	            // Check gaps is a routine that checks all the time if the gap and head to head distance is acording to the configuration.
	            // If not, the bit "sx_Gapping" is set true and the conveyor stops to gap.
	            // Compare gaps calculated with the configured gaps
	            IF NOT #sx_ReverseDirection
	            THEN
	                REGION 7.5.1 - Forward

	                    IF ((#sdi_GapHeadToHeadConfigurationFwd > #sdi_GapHeadToHeadFwd               // Compare head to head configured with real distance
	                        OR #sdi_GapTailToHeadConfigurationFwd > #sdi_GapFwd
	                        OR #sdi_GapTailToHeadConfigurationFwd > #sdi_DownstreamGapTailtoHeadFwd           // Compare gap configured with real gap
	                        OR #sdi_GapHeadToHeadConfigurationFwd > #sdi_DownstreamGapHeadToHeadFwd)
	                        AND #sF_TRIG_AuxHeadToEnd_Fwd.Q)                                                         // Trigger when parcel arrive in the end of the conveyor
	                    THEN

	                        #sx_GappingFwd := TRUE;        // Bit to inform the system that conveyor needs to stop to apply gap

	                    END_IF;

	                END_REGION
	            ELSE
	                REGION 7.5.1 - Reverse

	                    IF ((#sdi_GapHeadToHeadConfigurationRvs > #sdi_GapHeadToHeadRvs               // Compare head to head configured with real distance
	                        OR #sdi_GapTailToHeadConfigurationRvs > #sdi_Gap_Rvs
	                        OR #sdi_GapTailToHeadConfigurationRvs > #sdi_DownstreamGapTailtoHeadRvs           // Compare gap configured with real gap
	                        OR #sdi_GapHeadToHeadConfigurationRvs > #sdi_DownstreamGapHeadToHeadRvs)
	                        AND #sF_TRIG_AuxHeadToEnd_Rvs.Q)                                                         // Trigger when parcel arrive in the end of the conveyor
	                    THEN

	                        #sx_GappingRvs := TRUE;        // Bit to inform the system that conveyor needs to stop to apply gap

	                    END_IF;

	                END_REGION
	            END_IF;
	            //    When conveyor stops to gapping, displacement values from downstream are used to
	            //    apply new gap.
	            //    When the new gap applied fits with the configured one, the conveyor starts running again.
	            //    If the conveyor stops for die back reason and the gap its been applied, and extra gap value it will be applied.
	            //    This recovery gap it helps to recovery the system after die back.
	            IF NOT #sx_ReverseDirection
	            THEN
	                REGION 7.5.3 - Forward

	                    IF (#sx_GappingFwd          // Gapping needs to be applied bit
	                        AND ((#sdi_GapHeadToHeadConfigurationFwd > #sdi_GapHeadToHeadFwd    // Configured head to head bigger than the actual one
	                        OR #sdi_GapHeadToHeadConfigurationFwd - #idi_PECEoSDistance / 10 + #sdi_PECtoEndDistanceFwd > #sdi_DownstreamGapHeadToHeadFwd
	                        OR #sdi_GapTailToHeadConfigurationFwd > #sdi_GapFwd     // Configured gap bigger than the actual one
	                        OR #sdi_GapTailToHeadConfigurationFwd - #idi_PECEoSDistance / 10 + #sdi_PECtoEndDistanceFwd > #sdi_DownstreamGapTailtoHeadFwd)
	                        AND NOT #sx_RecoveryGapFwd)                                                // Die back recovery gap bit not active
	                        OR (((#sdi_GapHeadToHeadConfigurationFwd + #iUDT_ConveyorConfiguration.ExtraGapRecovery)   // Add recovery gap to the configured
	                        > #sdi_GapHeadToHeadFwd                                                                                 // Actual head to head distance
	                        OR (#sdi_GapHeadToHeadConfigurationFwd - #idi_PECEoSDistance / 10 + #sdi_PECtoEndDistanceFwd + #iUDT_ConveyorConfiguration.ExtraGapRecovery)
	                        > #sdi_DownstreamGapHeadToHeadFwd
	                        OR (#sdi_GapTailToHeadConfigurationFwd + #iUDT_ConveyorConfiguration.ExtraGapRecovery)    // Add recovery gap to the configured
	                        > #sdi_GapFwd                                                                               // Actual gap between parcels
	                        OR (#sdi_GapTailToHeadConfigurationFwd - #idi_PECEoSDistance / 10 + #sdi_PECtoEndDistanceFwd + #iUDT_ConveyorConfiguration.ExtraGapRecovery)
	                        > #sdi_DownstreamGapTailtoHeadFwd)
	                        AND #sx_RecoveryGapFwd))                                                                       // Recovery gap bit activate
	                    THEN

	                        #sdi_GapHeadToHeadFwd += #iqUDT_HandShake.DownstreamDisplacement;      // Increase head to head counter with conveyor downstream displacement
	                        #sdi_GapFwd += #iqUDT_HandShake.DownstreamDisplacement;     // Increase gap counter with conveyor downstream displacement

	                    ELSE

	                        #sx_GappingFwd := FALSE;                   // Set gapping bit to false

	                    END_IF;

	                    IF #sx_GappingFwd                              // Gapping bit active
	                        AND NOT #iqUDT_HandShake.RTR           // Ready to receive not active
	                    THEN

	                        #sx_RecoveryGapFwd := TRUE;                // Recovery gap activation after die back

	                    END_IF;

	                    IF #sx_RecoveryGapFwd                          // Recovery gap active
	                        AND NOT #sx_GappingFwd                     // Gapping bit not active
	                    THEN

	                        #sx_RecoveryGapFwd := FALSE;               // Recovery gap disable

	                    END_IF;

	                END_REGION
	            ELSE
	                REGION 7.5.4 - Reverse

	                    IF (#sx_GappingRvs          // Gapping needs to be applied bit
	                        AND ((#sdi_GapHeadToHeadConfigurationRvs > #sdi_GapHeadToHeadRvs    // Configured head to head bigger than the actual one
	                        OR #sdi_GapHeadToHeadConfigurationRvs - #idi_PECBoSDistance / 10 + #sdi_PECtoEndDistanceRvs > #sdi_DownstreamGapHeadToHeadRvs
	                        OR #sdi_GapTailToHeadConfigurationRvs > #sdi_Gap_Rvs     // Configured gap bigger than the actual one
	                        OR #sdi_GapTailToHeadConfigurationRvs - #idi_PECBoSDistance / 10 + #sdi_PECtoEndDistanceRvs > #sdi_DownstreamGapTailtoHeadRvs)
	                        AND NOT #sx_RecoveryGapRvs)                                                // Die back recovery gap bit not active
	                        OR (((#sdi_GapHeadToHeadConfigurationRvs + #iUDT_ConveyorConfiguration.ExtraGapRecovery)   // Add recovery gap to the configured
	                        > #sdi_GapHeadToHeadRvs                                                                                 // Actual head to head distance
	                        OR (#sdi_GapHeadToHeadConfigurationRvs - #idi_PECBoSDistance / 10 + #sdi_PECtoEndDistanceRvs + #iUDT_ConveyorConfiguration.ExtraGapRecovery)
	                        > #sdi_DownstreamGapHeadToHeadRvs
	                        OR (#sdi_GapTailToHeadConfigurationRvs + #iUDT_ConveyorConfiguration.ExtraGapRecovery)    // Add recovery gap to the configured
	                        > #sdi_Gap_Rvs                                                                               // Actual gap between parcels
	                        OR (#sdi_GapTailToHeadConfigurationRvs - #idi_PECBoSDistance / 10 + #sdi_PECtoEndDistanceRvs + #iUDT_ConveyorConfiguration.ExtraGapRecovery)
	                        > #sdi_DownstreamGapTailtoHeadRvs)
	                        AND #sx_RecoveryGapRvs))                                                                                // Recovery gap bit activate
	                    THEN

	                        #sdi_GapHeadToHeadRvs -= #iqUDT_HandShakeUp.DownstreamDisplacement;      // Increase head to head counter with conveyor downstream displacement
	                        #sdi_Gap_Rvs -= #iqUDT_HandShakeUp.DownstreamDisplacement;     // Increase gap counter with conveyor downstream displacement

	                    ELSE

	                        #sx_GappingRvs := FALSE;                   // Set gapping bit to false

	                    END_IF;

	                    IF #sx_GappingRvs                              // Gapping bit active
	                        AND NOT #iqUDT_HandShakeUp.RTR           // Ready to receive not active
	                    THEN

	                        #sx_RecoveryGapRvs := TRUE;                // Recovery gap activation after die back

	                    END_IF;

	                    IF #sx_RecoveryGapRvs                          // Recovery gap active
	                        AND NOT #sx_GappingRvs                     // Gapping bit not active
	                    THEN

	                        #sx_RecoveryGapRvs := FALSE;               // Recovery gap disable

	                    END_IF;

	                END_REGION
	            END_IF;
	        END_REGION

	        REGION 7.6 - Ready to send and Transfer in progress
	            IF NOT #sx_ReverseDirection
	            THEN
	                REGION 7.6.1 - Forward

	                    IF #iqUDT_HandShake.RTR                                            // Ready to receive bit
	                        AND NOT #sx_GappingFwd
	                        AND #sx_AuxHeadAtEndFwd                                            // Parcel is at end of conveyor
	                        AND NOT #ix_ExternalRequestDieBack
	                    THEN

	                        #iqUDT_HandShake.TIP := TRUE;      // Transfer in progress bit
	                        #iqUDT_HandShake.RTS := FALSE;     // Ready to send bit
	                        #sx_AuxHeadAtEndFwd := FALSE;

	                    END_IF;

	                    IF #sR_TRIG_TailToBegin_Fwd.Q               // Reset TIP when the parcel leaves interlock
	                    THEN

	                        #iqUDT_HandShake.TIP := FALSE;     // Transfer in progress bit

	                    END_IF;

	                END_REGION
	            ELSE
	                REGION 7.6.2 - Reverse

	                    IF #iqUDT_HandShakeUp.RTR                                            // Ready to receive bit
	                        AND #iqUDT_HandShake.RTR
	                        AND NOT #sx_GappingRvs
	                        AND #sx_AuxHeadAtEndRvs                                            // Parcel is at end of conveyor
	                        AND NOT #ix_ExternalRequestDieBack
	                    THEN

	                        #iqUDT_HandShakeUp.TIP := TRUE;      // Transfer in progress bit
	                        #iqUDT_HandShakeUp.RTS := FALSE;     // Ready to send bit
	                        #sx_AuxHeadAtEndRvs := FALSE;

	                    END_IF;

	                    IF #sR_TRIG_TailToBegin_Rvs.Q               // Reset TIP when the parcel leaves interlock
	                    THEN

	                        #iqUDT_HandShakeUp.TIP := FALSE;     // Transfer in progress bit

	                    END_IF;

	                END_REGION
	            END_IF;
	        END_REGION

	        REGION 7.7 - Downstream gap

	            (* This functionality is used to maintain the gap between parcel conveyor's downstream.
	               To do this, is used the downstream displacement.  *)
	            IF NOT #sx_ReverseDirection
	            THEN
	                REGION 7.7.1 - Forward

	                    IF #sR_TRIG_TailToBegin_Fwd.Q                       // When the parcel's tail reach the beginning of downstream conveyor
	                    THEN

	                        #sdi_DownstreamGapTailtoHeadFwd := 0;                     // Reset downstream gap counter

	                    END_IF;

	                    IF #sdi_DownstreamGapTailtoHeadFwd < #ci_OverflowLimit        // Prevent integer variable overflow
	                    THEN

	                        #sdi_DownstreamGapTailtoHeadFwd += #iqUDT_HandShake.DownstreamDisplacement;          // Downstream displacement gap counter

	                    END_IF;

	                END_REGION
	            ELSE
	                REGION 7.7.2 - Reverse

	                    IF #sR_TRIG_TailToBegin_Rvs.Q                       // When the parcel's tail reach the beginning of downstream conveyor
	                    THEN

	                        #sdi_DownstreamGapTailtoHeadRvs := 0;                     // Reset downstream gap counter

	                    END_IF;

	                    IF #sdi_DownstreamGapTailtoHeadRvs < #ci_OverflowLimit        // Prevent integer variable overflow
	                    THEN

	                        #sdi_DownstreamGapTailtoHeadRvs -= #iqUDT_HandShakeUp.DownstreamDisplacement;          // Downstream displacement gap counter

	                    END_IF;

	                END_REGION
	            END_IF;
	        END_REGION

	        REGION 7.8 - Downstream Head to Head
	            IF NOT #sx_ReverseDirection
	            THEN
	                REGION 7.8.1 - Forward

	                    #sR_TRIG_Transfering_Fwd(CLK := #iqUDT_HandShake.TIP);

	                    IF #sR_TRIG_Transfering_Fwd.Q                                                           // Transfering aux bit rising trigger
	                    THEN

	                        #sdi_DownstreamGapHeadToHeadFwd := 0;                                              // Downstream head to head reset counter

	                    END_IF;

	                    IF #sdi_DownstreamGapHeadToHeadFwd < #ci_OverflowLimit                                 // Prevent integer variable overflow
	                    THEN

	                        #sdi_DownstreamGapHeadToHeadFwd += #iqUDT_HandShake.DownstreamDisplacement;       // Downstream displacement head to head counter

	                    END_IF;

	                END_REGION
	            ELSE
	                REGION 7.8.2 - Reverse

	                    #sR_TRIG_Transfering_Rvs(CLK := #iqUDT_HandShake.TIP);

	                    IF #sR_TRIG_Transfering_Rvs.Q                                                           // Transfering aux bit rising trigger
	                    THEN

	                        #sdi_DownstreamGapHeadToHeadRvs := 0;                                              // Downstream head to head reset counter

	                    END_IF;

	                    IF #sdi_DownstreamGapHeadToHeadRvs < #ci_OverflowLimit                                 // Prevent integer variable overflow
	                    THEN

	                        #sdi_DownstreamGapHeadToHeadRvs -= #iqUDT_HandShakeUp.DownstreamDisplacement;       // Downstream displacement head to head counter

	                    END_IF;

	                END_REGION
	            END_IF;
	        END_REGION

	        REGION 7.9 - Energy save

	            (* Save energy functionality is used to stop conveyor if no parcels are in the system to save energy
	               Save energy function counts displacement if the photo eye do not detects parcels. The counter is reset if:
	               - Photo eye is triggered.
	               - Reset is required from external.
	               - Ready to send is active from upstream. *)

	            IF #iUDT_ConveyorConfiguration.Energy                                       // Energy save functionality enable from configuration
	            THEN

	                IF #sdi_AuxEnergySaveFwd >= #iUDT_ConveyorConfiguration.Forward_Direction.EnergySaveLenght        // Compare energy save counter with configured lenght
	                    OR #sdi_AuxEnergySaveRvs >= #iUDT_ConveyorConfiguration.Reverse_Direction.EnergySaveLenght
	                THEN
	                    #sx_EnergySaveActive := TRUE;                                           // Set energy save active true
	                END_IF;

	                IF ((NOT #ix_PECEoS OR NOT #ix_PECBoS)                                  // Photo eye detects a parcel
	                    AND NOT #sx_EnergySaveActive)                                         // Energy save active bit
	                    OR #ix_ResetEnergySave                                               // Reset energy save
	                    OR (#iqUDT_HandShakeUp.ResetEnergySave AND NOT #sx_ReverseDirection)                               // Reset energy save externaly
	                    OR (#iqUDT_HandShake.ResetEnergySave AND #sx_ReverseDirection)
	                    OR NOT #iqUDT_EquipmentControl.Command.AutomaticOn                  // Automatic ON from control block
	                    OR #iqUDT_EquipmentControl.Command.Stop                             // Stop command from control block
	                THEN
	                    #sdi_AuxEnergySaveFwd := 0;                                        // Reset energy save counter
	                    #sdi_AuxEnergySaveRvs := 0;                                        // Reset energy save counter
	                    #sx_EnergySaveActive := FALSE;                                      // Set energy save active to false
	                ELSE
	                    // Increament displacement counter
	                    IF NOT #sx_ReverseDirection
	                    THEN
	                        #sdi_AuxEnergySaveFwd += #iqUDT_ConveyorInterface.Displacement;
	                    ELSE
	                        #sdi_AuxEnergySaveRvs -= #iqUDT_ConveyorInterface.Displacement;
	                    END_IF;
	                END_IF;

	            ELSE
	                // If energy save functionality is disable from configuration
	                #sdi_AuxEnergySaveFwd := 0;                                             // Reset energy save counter
	                #sx_EnergySaveActive := FALSE;                                      // Set energy save false
	            END_IF;
	            // Reset to downstream when not already in enery save on signal of PEC
	            // When slave conveyor pass reset esave command to master conveyor

	            IF NOT #sx_ReverseDirection
	            THEN
	                #iqUDT_HandShake.ResetEnergySave := (NOT #ix_PECEoS OR #sx_AuxHeadAtEndFwd OR #iqUDT_HandShake.TIP) AND NOT #sx_EnergySaveActive
	                OR (#iUDT_ConveyorConfiguration.Forward_Direction.Mode = 1 AND #iqUDT_HandShakeUp.ResetEnergySave);
	            ELSE
	                #iqUDT_HandShakeUp.ResetEnergySave := NOT #ix_PECBoS AND NOT #sx_EnergySaveActive
	                OR (#iUDT_ConveyorConfiguration.Reverse_Direction.Mode = 1 AND #iqUDT_HandShake.ResetEnergySave);
	            END_IF;
	        END_REGION

	        REGION 7.10 - Operation modes

	            // Different modes in automatic can be configured
	            // 1 - Slave
	            // 2 - Queue
	            // 3 - Bulk flow

	            IF #sx_AutomaticActive                                          // Automatic mode active
	                AND #tx_CascadeStart                                        // Cascade startup
	            THEN

	                IF NOT #sx_ReverseDirection
	                THEN

	                    CASE #iUDT_ConveyorConfiguration.Forward_Direction.Mode OF                   // Operation mode configured

	                        1:  // Slave

	                            // Run conveyor if ready to receive if on, and conveyor is not gapping,
	                            // and not halt request and not energy save active

	                            #iqUDT_ConveyorInterface.RunFwd := #sx_AutomaticActive     // Automatic mode active
	                            AND #sx_Ready                                               // Ready active
	                            AND NOT #ix_ExternalRequestHold                             // Halt request is not active
	                            AND NOT #sx_EnergySaveActive                                // Energy save not active
	                            AND #iqUDT_HandShake.RTR                               // Ready to receive active
	                            AND NOT #sx_DirectionChanged;

	                            #iqUDT_HandShakeUp.RTR := #iqUDT_ConveyorInterface.RunFwd;

	                        2:  // Master

	                            // With queue configuration, conveyor runs if ready to receive is true.
	                            // If ready to receive is false, conveyor runs until parcel reach the end of the conveyor.

	                            // Conveyor stops if heads parcel reache the end of the conveyor and:
	                            // - Ready to receive is false
	                            // - Or die back requested.
	                            // - Or halt requested
	                            // Conveyor also stops if gapping is active or energy save mode active.

	                            #iqUDT_ConveyorInterface.RunFwd := #sx_AutomaticActive             // Automatic mode active
	                            AND #sx_Ready                                                       // Ready active
	                            AND NOT #sx_DirectionChanged
	                            AND NOT #sx_GappingFwd                                                 // Gapping request
	                            AND NOT #sx_EnergySaveActive                                        // Energy save request
	                            AND NOT #ix_ExternalRequestHold                                     // Halt requested from external
	                            AND ((NOT #ix_ExternalRequestDieBack
	                            AND #iqUDT_HandShake.RTR)
	                            OR (NOT #sx_AuxHeadAtEndFwd
	                            AND NOT #iqUDT_HandShake.TIP)
	                            OR (#iqUDT_HandShake.RTR
	                            AND NOT #sx_AuxHeadAtEndFwd));

	                            #iqUDT_HandShakeUp.RTR := #iqUDT_ConveyorInterface.RunFwd;


	                        3: //Master at bulk flow

	                            #iqUDT_ConveyorInterface.RunFwd := #sx_AutomaticActive             // Automatic mode active
	                            AND #sx_Ready                                                       // Ready active
	                            AND NOT #sx_DirectionChanged
	                            AND NOT #sx_EnergySaveActive                                        // Energy save request
	                            AND NOT #ix_ExternalRequestHold                                     // Halt requested from external
	                            AND (
	                            (NOT #ix_ExternalRequestDieBack                                     //no die back request and the downstream is running
	                            AND #iqUDT_HandShake.RTR)
	                            OR                                                                  //..or..
	                            (#sdi_TransitionZone = 0)                                            // no parcels at the transition zone
	                            OR                                                                  //..or..
	                            (#iqUDT_HandShake.RTR
	                            AND NOT #ix_ExternalRequestDieBack
	                            AND NOT (#sdi_TransitionZone = 0)));                                  //downstream is running and there are

	                            //If PEC is blocked, reset tracking counter
	                            IF NOT #ix_PECEoS THEN
	                                #sdi_TransitionZone := (#idi_PECEoSDistance / 10);
	                            END_IF;

	                            //Track parcels at the zone between EoS and conveyor end (Transition Zone)
	                            #sdi_TransitionZone := #sdi_TransitionZone - #iqUDT_ConveyorInterface.Displacement;

	                            //If Value is negative then set to 0
	                            IF #sdi_TransitionZone < 0 THEN
	                                #sdi_TransitionZone := 0;
	                            END_IF;

	                            #iqUDT_HandShakeUp.RTR := #iqUDT_ConveyorInterface.RunFwd;

	                    END_CASE;

	                ELSE

	                    CASE #iUDT_ConveyorConfiguration.Reverse_Direction.Mode OF                   // Operation mode configured

	                        1:  // Slave

	                            // Run conveyor if ready to receive if on, and conveyor is not gapping,
	                            // and not halt request and not energy save active

	                            #iqUDT_ConveyorInterface.RunRvs := #sx_AutomaticActive     // Automatic mode active
	                            AND #sx_Ready                                               // Ready active
	                            AND NOT #ix_ExternalRequestHold                             // Halt request is not active
	                            AND NOT #sx_EnergySaveActive                                // Energy save not active
	                            AND #iqUDT_HandShakeUp.RTR                                 // Ready to receive active
	                            AND NOT #sx_DirectionChanged;

	                            #iqUDT_HandShake.RTR := #iqUDT_ConveyorInterface.RunRvs;

	                        2:  // Master

	                            // With queue configuration, conveyor runs if ready to receive is true.
	                            // If ready to receive is false, conveyor runs until parcel reach the end of the conveyor.

	                            // Conveyor stops if heads parcel reache the end of the conveyor and:
	                            // - Ready to receive is false
	                            // - Or die back requested.
	                            // - Or halt requested
	                            // Conveyor also stops if gapping is active or energy save mode active.

	                            #iqUDT_ConveyorInterface.RunRvs := #sx_AutomaticActive             // Automatic mode active
	                            AND #sx_Ready                                                       // Ready active
	                            AND NOT #sx_DirectionChanged
	                            AND NOT #sx_GappingRvs                                             // Gapping request
	                            AND NOT #sx_EnergySaveActive                                        // Energy save request
	                            AND NOT #ix_ExternalRequestHold                                     // Halt requested from external
	                            AND ((NOT #ix_ExternalRequestDieBack
	                            AND #iqUDT_HandShakeUp.RTR)
	                            OR (NOT #sx_AuxHeadAtEndRvs
	                            AND NOT #iqUDT_HandShakeUp.TIP)
	                            OR (#iqUDT_HandShakeUp.RTR
	                            AND NOT #sx_AuxHeadAtEndRvs));

	                            #iqUDT_HandShake.RTR := #iqUDT_ConveyorInterface.RunRvs;


	                        3: //Master at bulk flow

	                            #iqUDT_ConveyorInterface.RunRvs := #sx_AutomaticActive             // Automatic mode active
	                            AND #sx_Ready                                                       // Ready active
	                            AND NOT #sx_DirectionChanged
	                            AND NOT #sx_EnergySaveActive                                        // Energy save request
	                            AND NOT #ix_ExternalRequestHold                                     // Halt requested from external
	                            AND (
	                            (NOT #ix_ExternalRequestDieBack                                     //no die back request and the downstream is running
	                            AND #iqUDT_HandShakeUp.RTR)
	                            OR                                                                  //..or..
	                            (#sdi_TransitionZone = 0)                                            // no parcels at the transition zone
	                            OR                                                                  //..or..
	                            (#iqUDT_HandShakeUp.RTR
	                            AND NOT #ix_ExternalRequestDieBack
	                            AND NOT (#sdi_TransitionZone = 0)));                                  //downstream is running and there are

	                            //If PEC is blocked, reset tracking counter
	                            IF NOT #ix_PECBoS THEN
	                                #sdi_TransitionZone := #idi_PECEoSDistance / 10;
	                            END_IF;
	                            //Track parcels at the zone between EoS and conveyor end (Transition Zone)
	                            #sdi_TransitionZone := #sdi_TransitionZone - #iqUDT_ConveyorInterface.Displacement;

	                            //If Value is negative then set to 0
	                            IF #sdi_TransitionZone < 0 THEN
	                                #sdi_TransitionZone := 0;
	                            END_IF;

	                            #iqUDT_HandShake.RTR := #iqUDT_ConveyorInterface.RunRvs;
	                    END_CASE;

	                END_IF;

	            ELSE

	                // If conveyor is not in manual mode and not ready
	                IF NOT #sx_ReverseDirection
	                THEN
	                    #iqUDT_ConveyorInterface.RunFwd := FALSE;                      // Order to VFD stop conveyor
	                    #iqUDT_HandShakeUp.RTR := FALSE;                               // Set ready to receive false
	                ELSE
	                    #iqUDT_ConveyorInterface.RunRvs := FALSE;                      // Order to VFD stop conveyor
	                    #iqUDT_HandShake.RTR := FALSE;                               // Set ready to receive false
	                END_IF;

	            END_IF;

	        END_REGION

	    END_IF;
	END_REGION

	REGION 8 - Speed control

	    (*In manual mode, conveyor default runs with manual speed which is calculated as a percentage of nominal speed. If "ManualFullSpeed" is set true, conveyor runs with high speed in manual mode.
	     In jog mode conveyor always runs in low speed. In automatic mode, conveyor runs with full speed if external is zero. If external speed is bigger than zero, conveyor will run with that speed. *)


	    // security
	    IF #iqUDT_ConveyorCommand.ManualSpeed > 100 THEN
	        #iqUDT_ConveyorCommand.ManualSpeed := 100;
	    END_IF;

	    IF #iqUDT_ConveyorCommand.ManualSpeed < 0 THEN
	        #iqUDT_ConveyorCommand.ManualSpeed := 0;
	    END_IF;



	    IF #sx_ManualModeActive                                                                         // Manual mode active
	    THEN

	        IF #iqUDT_ConveyorCommand.ManualStartStop                                              // Full speed in manual mode
	        THEN

	            IF #iqUDT_ConveyorCommand.ManualFullSpeed                                                  // Full speed in manual mode
	            THEN
	                #iqUDT_ConveyorInterface.SpeedSetpoint := #iUDT_ConveyorConfiguration.SpeedSetpointNominal;    // Move nominal setpoint to the VDF

	            ELSE
	                #iqUDT_ConveyorInterface.SpeedSetpoint := REAL_TO_INT(INT_TO_REAL(#iqUDT_ConveyorCommand.ManualSpeed) * (INT_TO_REAL(#iUDT_ConveyorConfiguration.SpeedSetpointNominal) / 100));     // Calculate and Move manual speed setpoint to VFD

	            END_IF;

	        ELSE                                                                                             //low speed for jog mode

	            IF #iUDT_ConveyorConfiguration.SpeedSetpointLow < #iUDT_ConveyorConfiguration.SpeedSetpointNominal  //Low speed can't be higher than nominal speed
	            THEN
	                #iqUDT_ConveyorInterface.SpeedSetpoint := #iUDT_ConveyorConfiguration.SpeedSetpointLow;    // Move low speed setpoint to the VDF

	            ELSE

	                #iqUDT_ConveyorInterface.SpeedSetpoint := #iUDT_ConveyorConfiguration.SpeedSetpointNominal;    // Move low speed setpoint to the VDF
	            END_IF;
	        END_IF;



	    ELSE

	        IF #ii_ExternalSpeed > 0                                                                      // If external speed bigger than zero
	        THEN
	            #iqUDT_ConveyorInterface.SpeedSetpoint := #ii_ExternalSpeed;                                     // Move external speed to VFD
	        ELSE
	            #iqUDT_ConveyorInterface.SpeedSetpoint := #iUDT_ConveyorConfiguration.SpeedSetpointNominal;       // Move nominal setpoint to VFD
	        END_IF;

	    END_IF;



	END_REGION


	REGION 9 - Status
	    #sUDT_HMIStatus.Specific.Reverse := #sx_ReverseDirection;

	    // stopped
	    #sUDT_CommonStatus.Stopped := NOT #sx_Ready OR NOT #sx_AutomaticActive;

	    // Auto ON
	    #sUDT_CommonStatus.AutoON := #sx_Ready AND #sx_AutomaticActive;

	    // Running
	    #sUDT_CommonStatus.Running := #iqUDT_ConveyorInterface.RunFwd
	    OR #iqUDT_ConveyorInterface.RunRvs;

	    // Halted
	    #sUDT_CommonStatus.Halted := #ix_ExternalRequestHold
	    AND #sUDT_CommonStatus.AutoON
	    AND NOT #sUDT_CommonStatus.EnergySave;

	    // Energy save active
	    #sUDT_CommonStatus.EnergySave := #sx_EnergySaveActive AND #sx_AutomaticActive;

	    // Die back
	    #sUDT_CommonStatus.Dieback := #sUDT_CommonStatus.AutoON
	    AND NOT #sUDT_CommonStatus.EnergySave
	    AND NOT #sUDT_CommonStatus.Running;

	    // Manual
	    #sUDT_CommonStatus.Manual := #sx_ManualModeActive;

	    // Manual Running
	    #sUDT_CommonStatus.ManualRun := #sx_ManualModeActive AND #sUDT_CommonStatus.Running;

	    // Safety not ok
	    #sUDT_CommonStatus.SafetyStop := NOT #ix_SafetyOk AND #ix_HardwareOk;

	    // HMI status update
	    IF #sUDT_CommonStatusOld <> #sUDT_CommonStatus                                            // update on change
	        OR (#sR_TRIG_Reverse.Q OR #sF_TRIG_Reverse.Q)
	    THEN
	        // HMI status initialization
	        #sUDT_HMIStatus.Status := 0;

	        // Energy save
	        IF #sUDT_CommonStatus.EnergySave
	        THEN
	            #sUDT_HMIStatus.Status := "DB_HMIStatusConfiguration".EnergySave;
	        END_IF;

	        // Running
	        IF #sUDT_CommonStatus.Running
	        THEN
	            #sUDT_HMIStatus.Status := "DB_HMIStatusConfiguration".Running;
	        END_IF;

	        // Stopped
	        IF #sUDT_CommonStatus.Stopped
	        THEN
	            #sUDT_HMIStatus.Status := "DB_HMIStatusConfiguration".Stopped;
	        END_IF;

	        // Dieback
	        IF #sUDT_CommonStatus.Dieback
	        THEN
	            #sUDT_HMIStatus.Status := "DB_HMIStatusConfiguration".Dieback;
	        END_IF;

	        // Halted
	        IF #sUDT_CommonStatus.Halted
	        THEN
	            #sUDT_HMIStatus.Status := "DB_HMIStatusConfiguration".Halted;
	        END_IF;

	        // Manual
	        IF #sUDT_CommonStatus.Manual
	        THEN
	            #sUDT_HMIStatus.Status := "DB_HMIStatusConfiguration".Manual;
	        END_IF;

	        // Running in manual mode
	        IF #sUDT_CommonStatus.ManualRun
	        THEN
	            #sUDT_HMIStatus.Status := "DB_HMIStatusConfiguration".ManualRun;
	        END_IF;

	(*        // Internal tracking warning
	        IF #iq_UDT_ConveyorInterface.InternalWarningTracking
	        THEN
	            #s_UDT_HMIStatus.Status := "DB_HMIStatusConfiguration".Warning;
	        END_IF; *)

	        // Internal tracking error
	        IF #iqUDT_ConveyorInterface.InternalErrorTracking
	        THEN
	            #sUDT_HMIStatus.Status := "DB_HMIStatusConfiguration".TrackingError;
	        END_IF;

	        // Internal PEC error
	        IF #iqUDT_ConveyorInterface.InternalErrorPEC
	        THEN
	            #sUDT_HMIStatus.Status := "DB_HMIStatusConfiguration".PECJam;
	        END_IF;

	        // Internal Encoder error
	        IF #iqUDT_ConveyorInterface.InternalErrorEncoder
	        THEN
	            #sUDT_HMIStatus.Status := "DB_HMIStatusConfiguration".EncoderError;
	        END_IF;

	        // Internal VFD error
	        IF #iqUDT_ConveyorInterface.InternalErrorVFD
	        THEN
	            #sUDT_HMIStatus.Status := "DB_HMIStatusConfiguration".VFDError;
	        END_IF;

	        // Disconnect error
	        IF #iqUDT_ConveyorInterface.Disconnected
	        THEN
	            #sUDT_HMIStatus.Status := "DB_HMIStatusConfiguration".CBError;
	        END_IF;

	        // Safety stop
	        IF (#sUDT_CommonStatus.SafetyStop)
	        THEN
	            #sUDT_HMIStatus.Status := "DB_HMIStatusConfiguration".SafetyStop;
	        END_IF;

	        #sUDT_CommonStatusOld := #sUDT_CommonStatus;              // Copy status to memory
	        #qUDT_Status := #sUDT_CommonStatus;                       // Copy status to output

	    END_IF;

	    // Copy HMI status to output
	    #qUDT_HMIStatus := #sUDT_HMIStatus;

	END_REGION


	REGION 10 - Statistics

	    REGION 10.1 - Conveyor up time

	        IF #sx_Up OR #iqUDT_EquipmentControl.Command.ResetData    // Reset statistics
	        THEN

	            "FC_Statistics"(ix_Reset := #iqUDT_EquipmentControl.Command.ResetData,      // Reset statistics input
	                            ix_Activate := #sx_Up,
	                            ix_RTrigActivate := #sR_TRIG_ConveyorUp.Q,                     // Statistics active trigger
	                            iqUDT_Statistics := #iqUDT_Statistics.ConveyorUp);      // Statistics values output

	        END_IF;

	    END_REGION

	    REGION 10.2 - Energy save

	        // Statistics Energy save mode active
	        IF #sUDT_CommonStatus.EnergySave(* #sx_EnergySaveActive *)                                                        // Energy save active
	            OR #iqUDT_EquipmentControl.Command.ResetData                               // Reset statistics
	        THEN
	            "FC_Statistics"(ix_Reset := #iqUDT_EquipmentControl.Command.ResetData,      // Reset statistics input
	                            ix_Activate := #sUDT_CommonStatus.EnergySave,                         // Activate statistics functions input
	                            ix_RTrigActivate := #sR_TRIG_EnergySave.Q,                    // Statistics active trigger
	                            iqUDT_Statistics := #iqUDT_Statistics.EnergySave);         // Statistics values output

	        END_IF;

	    END_REGION

	    REGION 10.3 - Conveyor down time

	        // Conveyor down is when conveyor is not in manual mode and has an error
	        IF #sx_Down OR #iqUDT_EquipmentControl.Command.ResetData OR #sUDT_CommonStatus.SafetyStop                                    // Reset statistics
	        THEN

	            "FC_Statistics"(ix_Reset := #iqUDT_EquipmentControl.Command.ResetData,             // Reset statistics input
	                            ix_Activate := #sx_Down OR #sUDT_CommonStatus.SafetyStop, // Activate statistics functions input
	                            ix_RTrigActivate := #sR_TRIG_ConveyorDownTime.Q,                     // Statistics active trigger
	                            iqUDT_Statistics := #iqUDT_Statistics.ConveyorDown);              // Statistics values output

	        END_IF;
	    END_REGION

	    REGION 10.4 - Conveyor stop time

	        IF #sx_Stopped OR #iqUDT_EquipmentControl.Command.ResetData                                           // Reset statistics
	        THEN

	            "FC_Statistics"(ix_Reset := #iqUDT_EquipmentControl.Command.ResetData,        // Reset statistics input
	                            ix_Activate := #sx_Stopped,                                           // Activate statistics functions input
	                            ix_RTrigActivate := #sR_TRIG_ConveyorStopped.Q,                        // Statistics active trigger
	                            iqUDT_Statistics := #iqUDT_Statistics.ConveyorStop);                  // Statistics values output

	        END_IF;
	    END_REGION

	END_REGION

	REGION 11 - Report to control block
	    // Function to manage report between control block and conveyor block
	    "FC_EquipmentReport"(iUDT_Status := #sUDT_CommonStatus,
	                         iqUDT_Control := #iqUDT_EquipmentControl);

	END_REGION

	REGION 12 - Internal errors and warnings reset

	    IF #iqUDT_EquipmentControl.Command.Reset
	    THEN

	        #iqUDT_ConveyorInterface.InternalErrorEncoder := FALSE;
	        #iqUDT_ConveyorInterface.InternalErrorPEC := FALSE;
	        #iqUDT_ConveyorInterface.InternalWarningTracking := FALSE;
	        #iqUDT_ConveyorInterface.InternalErrorTracking := FALSE;
	        #iqUDT_ConveyorInterface.InternalWarningVFD := FALSE;
	        #iqUDT_ConveyorInterface.InternalErrorVFD := FALSE;
	        #iqUDT_ConveyorInterface.Disconnected := FALSE;
	        #iqUDT_ConveyorInterface.ConfigurationError := FALSE;
	    END_IF;

	END_REGION

END_FUNCTION_BLOCK

FUNCTION_BLOCK "FB_DimensionsCheck"
{ S7_Optimized_Access := 'TRUE' }
VERSION : 0.1
// ATTRIBUTES
// AUTO_NUMBER = True
// BLOCK_NUMBER = 208
// END_ATTRIBUTES
   VAR_INPUT
      iUDT_DimensionsCheckConfiguration { ExternalAccessible := 'False'; ExternalVisible := 'False'; ExternalWritable := 'False'} : "UDT_DimensionsCheckConfiguration";   //    Dimensions check configuration structure
      ix_LenghtPEC1 { ExternalAccessible := 'False'; ExternalVisible := 'False'; ExternalWritable := 'False'} : Bool;   //    Length 1  PEC
      ix_LenghtPEC2 { ExternalAccessible := 'False'; ExternalVisible := 'False'; ExternalWritable := 'False'} : Bool;   //    Length 2 PEC
      ix_HeightPEC { ExternalAccessible := 'False'; ExternalVisible := 'False'; ExternalWritable := 'False'} : Bool;   //    Height PEC
      ix_WidthPEC { ExternalAccessible := 'False'; ExternalVisible := 'False'; ExternalWritable := 'False'} : Bool;   //    Width  PEC
      ix_Reset { ExternalAccessible := 'False'; ExternalVisible := 'False'; ExternalWritable := 'False'} : Bool;   //   TRUE when reset errors or reset energy save required
      ix_ReverseRun { ExternalAccessible := 'False'; ExternalVisible := 'False'; ExternalWritable := 'False'} : Bool;   //   TRUE when run conveyor in reverse direction is required
      ix_ResetStatistics { ExternalAccessible := 'False'; ExternalVisible := 'False'; ExternalWritable := 'False'} : Bool;   //   TRUE when reset statistics required
      ix_ConveyorEsaveStatus { ExternalAccessible := 'False'; ExternalVisible := 'False'; ExternalWritable := 'False'} : Bool;   // Conveyor Energy save Status: In Esave
      ix_HardwareOK { ExternalAccessible := 'False'; ExternalVisible := 'False'; ExternalWritable := 'False'} : Bool;   // TRUE when 24V on RIO with DMC signals is OK
   END_VAR

   VAR_OUTPUT
      qUDT_HMIStatus { ExternalAccessible := 'False'; ExternalVisible := 'False'; ExternalWritable := 'False'} : "UDT_DimensionsCheckStatus";   //    Dimensions check status error structure
      qx_Lamp { ExternalAccessible := 'False'; ExternalVisible := 'False'; ExternalWritable := 'False'} : Bool;   //    TRUE when lamp requested
      qx_ButtonLamp { ExternalAccessible := 'False'; ExternalVisible := 'False'; ExternalWritable := 'False'} : Bool;   //  Button lamp
      qx_Halt { ExternalAccessible := 'False'; ExternalVisible := 'False'; ExternalWritable := 'False'} : Bool;   //    TRUE when conveyor halt
      qx_WakeUp { ExternalAccessible := 'False'; ExternalVisible := 'False'; ExternalWritable := 'False'} : Bool;   //    TRUE when reset enery save mode requested
      qx_RunReverse { ExternalAccessible := 'False'; ExternalVisible := 'False'; ExternalWritable := 'False'} : Bool;   //    TRUE when conveyor run in reverse direction
   END_VAR

   VAR_IN_OUT
      iqUDT_DimensionsCheckStatistics : "UDT_DimensionsCheckStatistics";   //    Dimensions check statistics
      iqUDT_EquipmentControl : "UDT_EquipmentControl";   //  Equipment control structure
      iqUDT_ConveyorInterface : "UDT_ConveyorInterface";   // Conveyor interface structure
   END_VAR

   VAR
      sFB_HardwareOKSignalDelay { ExternalAccessible := 'False'; ExternalVisible := 'False'; ExternalWritable := 'False'; S7_SetPoint := 'False'} : "FB_TimerOnOffDelay";
      sFB_FirstLengthPECTimerOnOffDelay { ExternalAccessible := 'False'; ExternalVisible := 'False'; ExternalWritable := 'False'; S7_SetPoint := 'False'} : "FB_TimerOnOffDelay";   //    Length PEC 1 filter
      sFB_SecLengthPECTimerOnOffDelay { ExternalAccessible := 'False'; ExternalVisible := 'False'; ExternalWritable := 'False'; S7_SetPoint := 'False'} : "FB_TimerOnOffDelay";   //    Length PEC 2 filter
      sFB_HeightPECTimerOnOffDelay { ExternalAccessible := 'False'; ExternalVisible := 'False'; ExternalWritable := 'False'; S7_SetPoint := 'False'} : "FB_TimerOnOffDelay";   //    Heigh PEC filter
      sFB_Width1PECTimerOnOffDelay { ExternalAccessible := 'False'; ExternalVisible := 'False'; ExternalWritable := 'False'; S7_SetPoint := 'False'} : "FB_TimerOnOffDelay";   //    Width PEC 1 filter
      sFB_Width2PECTimerOnOffDelay { ExternalAccessible := 'False'; ExternalVisible := 'False'; ExternalWritable := 'False'; S7_SetPoint := 'False'} : "FB_TimerOnOffDelay";   //    Width PEC 2 filter
      sR_TRIG_ParcelTooLong {InstructionName := 'R_TRIG'; LibVersion := '1.0'; ExternalAccessible := 'False'; ExternalVisible := 'False'; ExternalWritable := 'False'; S7_SetPoint := 'False'} : R_TRIG;   //    Rising edge trigger of parcel too long error
      sR_TRIG_ParcelTooHigh {InstructionName := 'R_TRIG'; LibVersion := '1.0'; ExternalAccessible := 'False'; ExternalVisible := 'False'; ExternalWritable := 'False'; S7_SetPoint := 'False'} : R_TRIG;   //    Rising edge trigger of parcel too long error
      sR_TRIG_ParcelTooWide {InstructionName := 'R_TRIG'; LibVersion := '1.0'; ExternalAccessible := 'False'; ExternalVisible := 'False'; ExternalWritable := 'False'; S7_SetPoint := 'False'} : R_TRIG;   //    Rising edge trigger of parcel too wide trigger
      sR_TRIG_WidthPEC {InstructionName := 'R_TRIG'; LibVersion := '1.0'; ExternalAccessible := 'False'; ExternalVisible := 'False'; ExternalWritable := 'False'; S7_SetPoint := 'False'} : R_TRIG;   //    Detect parcel on the Width 1 PEC
      sUDT_Status { ExternalAccessible := 'False'; ExternalVisible := 'False'; ExternalWritable := 'False'; S7_SetPoint := 'False'} : "UDT_DimensionsCheckStatus";   //    Dimension check status structure
      sui_ActualParcelLenght { ExternalAccessible := 'False'; ExternalVisible := 'False'; ExternalWritable := 'False'} : DInt;   //    Actual parcel lenght
      sui_LengthPEC2Displacement { ExternalAccessible := 'False'; ExternalVisible := 'False'; ExternalWritable := 'False'} : DInt;   // displacement of the parcel after length pec trigger
      sui_widthPECDisplacement { ExternalAccessible := 'False'; ExternalVisible := 'False'; ExternalWritable := 'False'} : DInt;   // displacement of the parcel after width pec trigger
      si_1stPackageDistance { ExternalAccessible := 'False'; ExternalVisible := 'False'; ExternalWritable := 'False'} : Int;   //    Distance traveled by the first package after hitting the first Width PEC
      si_2ndPackageDistance { ExternalAccessible := 'False'; ExternalVisible := 'False'; ExternalWritable := 'False'} : Int;   //    Distance traveled by the second package after hitting the first Width PEC
      si_SickDistance1 { ExternalAccessible := 'False'; ExternalVisible := 'False'; ExternalWritable := 'False'} : Int;   //  Distance from the SICK1 [cm]
      si_SickDistance2 { ExternalAccessible := 'False'; ExternalVisible := 'False'; ExternalWritable := 'False'} : Int;   //  Distance from the SICK2 [cm]
      si_ParcelTooWideDisplacement { ExternalAccessible := 'False'; ExternalVisible := 'False'; ExternalWritable := 'False'} : Int;   // Displacement of the parcel
      sx_ConfigurationError { ExternalAccessible := 'False'; ExternalVisible := 'False'; ExternalWritable := 'False'} : Bool;   //    Configuration error
      sx_FirstLengthPEC_Filtered { ExternalAccessible := 'False'; ExternalVisible := 'False'; ExternalWritable := 'False'} : Bool;   //    Filtered signal of Length 1 PEC
      sx_SecLengthPEC_Filtered { ExternalAccessible := 'False'; ExternalVisible := 'False'; ExternalWritable := 'False'} : Bool;   //    Filtered signal of Length 2 PEC
      sx_HeightPEC_Filtered { ExternalAccessible := 'False'; ExternalVisible := 'False'; ExternalWritable := 'False'} : Bool;   //    Filtered signal of Heigth PEC
      sx_Width1PEC_Filtered { ExternalAccessible := 'False'; ExternalVisible := 'False'; ExternalWritable := 'False'} : Bool;   //    Filtered signal of Width 1 PEC
      sx_Width2PEC_Filtered { ExternalAccessible := 'False'; ExternalVisible := 'False'; ExternalWritable := 'False'} : Bool;   //    Filtered signal of Width 2 PEC
      sx_Halt { ExternalAccessible := 'False'; ExternalVisible := 'False'; ExternalWritable := 'False'} : Bool;   //    Static variable for halt conveyor
      sx_Lamp { ExternalAccessible := 'False'; ExternalVisible := 'False'; ExternalWritable := 'False'} : Bool;   //    Static variable for lamp control
      sx_WakeUp { ExternalAccessible := 'False'; ExternalVisible := 'False'; ExternalWritable := 'False'} : Bool;   //    Static variable for wake up from energy save signal
      sx_RunReverse { ExternalAccessible := 'False'; ExternalVisible := 'False'; ExternalWritable := 'False'} : Bool;   //    Run reverse request
      sx_Count1stDistance { ExternalAccessible := 'False'; ExternalVisible := 'False'; ExternalWritable := 'False'} : Bool;   //    Request to count distance traveled by parcel after hitting width 1 PEC
      sx_Count2ndDistance { ExternalAccessible := 'False'; ExternalVisible := 'False'; ExternalWritable := 'False'} : Bool;   //    Request to count distance traveled by parcel after hitting width 1 PEC in case where there is already another package between PECs
   END_VAR


BEGIN
	(*
	----------------------------------------------------------------------------------------

	Version history:
	Date        | Version   | Author        | Remark
	----------------------------------------------------------------------------------------
	23/10/2019  | 3.0       | J.Krawczuk    | Initial version
	13/03/2020  | 3.1       | A.Nowak       | Change the too long width detection and variables
	16/03/2020  | 3.2       | M.Kurpiers    | Adapting reviews
	27/08/2020  | 3.3       | A.Nowak       | Add status number creating
	31/08/2020  | 3.4       | A.Nowak       | Change reset of the too wide parcel status
	09/09/2021  | 3.5       | N.Kadam       | Change for Fedex Milano
	01/02/2022  | 3.6       | M.Piela       | Change signaling lamp into solid light when the parcel is too long
	16/03/2022  | 3.7       | M.Piela       | Width check fix
	16/05/2022  | 3.8       | M.Kurpiers    | ABS added to package length calculation
	17/06/2022  | 3.9       | M.Kurpiers    | HMI status initialization added
	19/07/2022  | 3.10      | M.Kurpiers    | Check if downstream conveyor is not running reverse during too wide check
	29/07/2022  | 3.10      | M.Piela       | Check heigth pec only when conveyor is running
	21/02/2023  | 4.0       | F.Baten       | 4.0 Release TIA 17.5
	*)

	REGION 1 - Triggers

	    // Preparing triggers for statistics.
	    #sR_TRIG_ParcelTooLong(CLK := #sUDT_Status.Specific.ParcelTooLong);
	    #sR_TRIG_ParcelTooHigh(CLK := #sUDT_Status.Specific.ParcelTooHigh);
	    #sR_TRIG_ParcelTooWide(CLK := #sUDT_Status.Specific.ParcelTooWide);

	END_REGION

	REGION 2 - 24v OK signal delay

	    #sFB_HardwareOKSignalDelay(iudi_OnDelayTime := 5000,
	                               ix_SignalToDelay := #ix_HardwareOK);

	END_REGION

	REGION 2 - Photo eye's filters

	    // First length check photo eye filter.
	    #sFB_FirstLengthPECTimerOnOffDelay(iudi_OffDelayTime := #iUDT_DimensionsCheckConfiguration.PECLength1OnTime,
	                                       iudi_OnDelayTime := #iUDT_DimensionsCheckConfiguration.PECLength1OffTime,
	                                       ix_Enable := TRUE,
	                                       ix_SignalToDelay := NOT #ix_LenghtPEC1,
	                                       qx_DelayedSignal => #sx_FirstLengthPEC_Filtered);
	    // Second length check photo eye filter.
	    #sFB_SecLengthPECTimerOnOffDelay(iudi_OnDelayTime := #iUDT_DimensionsCheckConfiguration.PECLength2OnTime,
	                                     iudi_OffDelayTime := #iUDT_DimensionsCheckConfiguration.PECLength2OffTime,
	                                     ix_SignalToDelay := NOT #ix_LenghtPEC2,
	                                     ix_Enable := TRUE,
	                                     qx_DelayedSignal => #sx_SecLengthPEC_Filtered);
	    // High check photo eye filter.
	    #sFB_HeightPECTimerOnOffDelay(iudi_OnDelayTime := #iUDT_DimensionsCheckConfiguration.PECHeightTimeOn,
	                                  iudi_OffDelayTime := #iUDT_DimensionsCheckConfiguration.PECHeightTimeOff,
	                                  ix_SignalToDelay := NOT #ix_HeightPEC,
	                                  ix_Enable := TRUE,
	                                  qx_DelayedSignal => #sx_HeightPEC_Filtered);
	    // Width 1 check photo eye filter.
	    #sFB_Width1PECTimerOnOffDelay(iudi_OnDelayTime := #iUDT_DimensionsCheckConfiguration.PECWidthOnTime,
	                                  iudi_OffDelayTime := #iUDT_DimensionsCheckConfiguration.PECWidthOffTime,
	                                  ix_SignalToDelay := NOT #ix_WidthPEC,
	                                  ix_Enable := TRUE,
	                                  qx_DelayedSignal => #sx_Width1PEC_Filtered);

	END_REGION

	REGION 3 - Error reset

	    // Reseting errors.
	    IF #ix_Reset
	    THEN
	        #sUDT_Status.Specific.ParcelTooHigh := FALSE;
	        #sUDT_Status.Specific.ParcelTooLong := FALSE;

	        IF NOT #sx_Width1PEC_Filtered
	        THEN
	            #sUDT_Status.Specific.ParcelTooWide := FALSE;
	        END_IF;
	    END_IF;

	    // Reseting conveyor energy save mode.
	    #sx_WakeUp := #ix_Reset;

	END_REGION

	REGION 4 - Configuration check

	    #sx_ConfigurationError :=
	    #iUDT_DimensionsCheckConfiguration.DistanceBetweenLenghtPECs <= 0
	    OR #iUDT_DimensionsCheckConfiguration.PECWidthCheckLimit <= 0;

	END_REGION

	REGION 5 - Package length calculation

	    // When first lenght check PEC is active displacement is added to actual parcel lenght.
	    IF #sx_FirstLengthPEC_Filtered
	    THEN
	        #sui_ActualParcelLenght += ABS(#iqUDT_ConveyorInterface.Displacement);
	        // When parcel leaves the first PEC then actual parcel lenght is reset.
	    ELSE
	        #sui_ActualParcelLenght := 0;
	    END_IF;

	END_REGION

	REGION 6 - Length check PEC long parcel detection

	    // If Length 2 PEC  is triggered for more than configured distance then set too long parcel error

	    IF #sx_SecLengthPEC_Filtered
	        AND #iqUDT_ConveyorInterface.RunFwd
	    THEN
	        #sui_LengthPEC2Displacement += ABS(#iqUDT_ConveyorInterface.Displacement);
	    ELSE
	        #sui_LengthPEC2Displacement := 0;
	    END_IF;

	    IF #sui_LengthPEC2Displacement > #iUDT_DimensionsCheckConfiguration.PECLength2CheckLimit
	    THEN
	        #sUDT_Status.Specific.ParcelTooLong := TRUE;
	    END_IF;

	END_REGION

	REGION 6 - Too long parcel detection

	    // Too long parcel error is set only when two length check PECs are covered by parcel and actual parcel lenght is greater than the distance between the Length PECs.
	    // If configured distance between two PECs is 0 then length check is disabled.
	    IF #iUDT_DimensionsCheckConfiguration.DistanceBetweenLenghtPECs > 0
	        AND #sx_SecLengthPEC_Filtered
	        AND #sx_FirstLengthPEC_Filtered
	        AND #sui_ActualParcelLenght > (#iUDT_DimensionsCheckConfiguration.DistanceBetweenLenghtPECs - #iUDT_DimensionsCheckConfiguration.ParcelLengthAllowedDeviation)
	        AND #sFB_HardwareOKSignalDelay.qx_DelayedSignal
	    THEN
	        #sUDT_Status.Specific.ParcelTooLong := TRUE;
	    END_IF;

	END_REGION

	REGION 7 - Too high parcel detection

	    IF #sx_HeightPEC_Filtered
	        AND #sFB_HardwareOKSignalDelay.qx_DelayedSignal
	        AND #iqUDT_ConveyorInterface.RunFwd
	    THEN
	        #sUDT_Status.Specific.ParcelTooHigh := TRUE;
	    END_IF;

	END_REGION

	REGION 8 - Too wide parcel detection

	    // When width detection check PEC is active then displacement is added to actual parcel lenght.
	    IF #sx_Width1PEC_Filtered AND NOT #iqUDT_ConveyorInterface.RunRvs
	    THEN
	        #sui_widthPECDisplacement += ABS(#iqUDT_ConveyorInterface.Displacement);
	        // When parcel leaves the PEC then actual parcel lenght is reset.
	    ELSE
	        #sui_widthPECDisplacement := 0;
	    END_IF;

	    IF #sui_widthPECDisplacement > #iUDT_DimensionsCheckConfiguration.PECWidthCheckLimit
	    THEN
	        #sUDT_Status.Specific.ParcelTooWide := TRUE;
	    END_IF;

	END_REGION

	REGION 9 - Halt request and lamp handling

	    IF #sUDT_Status.Specific.ParcelTooHigh
	        OR #sUDT_Status.Specific.ParcelTooWide
	        OR #sUDT_Status.Specific.ParcelTooLong
	    THEN
	        #sx_RunReverse := #ix_ReverseRun;
	        #sx_Halt := NOT #sx_RunReverse;
	        #sx_Lamp := TRUE;
	    END_IF;

	    IF NOT #sUDT_Status.Specific.ParcelTooHigh
	        AND NOT #sUDT_Status.Specific.ParcelTooLong
	        AND NOT #sUDT_Status.Specific.ParcelTooWide
	    THEN
	        #sx_Halt := FALSE;
	        #sx_Lamp := FALSE;
	        #sx_RunReverse := FALSE;
	    END_IF;

	END_REGION

	REGION 10 - Statistics

	    REGION 10.1 - Too long parcels statistics

	        IF #sUDT_Status.Specific.ParcelTooLong
	            OR #ix_ResetStatistics
	        THEN
	            "FC_Statistics"(ix_Reset := #ix_ResetStatistics,
	                            ix_Activate := #sUDT_Status.Specific.ParcelTooLong,
	                            ix_RTrigActivate := #sR_TRIG_ParcelTooLong.Q,
	                            iqUDT_Statistics := #iqUDT_DimensionsCheckStatistics.TooLongParcels);
	        END_IF;

	    END_REGION

	    REGION 10.2 - Too high parcels statistics

	        IF #sUDT_Status.Specific.ParcelTooHigh
	            OR #ix_ResetStatistics
	        THEN
	            "FC_Statistics"(ix_Reset := #ix_ResetStatistics,
	                            ix_Activate := #sUDT_Status.Specific.ParcelTooHigh,
	                            ix_RTrigActivate := #sR_TRIG_ParcelTooHigh.Q,
	                            iqUDT_Statistics := #iqUDT_DimensionsCheckStatistics.TooHighParcels);
	        END_IF;

	    END_REGION

	    REGION 10.3 - Too wide parcels statistics

	        IF #sUDT_Status.Specific.ParcelTooWide
	            OR #ix_ResetStatistics
	        THEN
	            "FC_Statistics"(ix_Reset := #ix_ResetStatistics,
	                            ix_Activate := #sUDT_Status.Specific.ParcelTooWide,
	                            ix_RTrigActivate := #sR_TRIG_ParcelTooWide.Q,
	                            iqUDT_Statistics := #iqUDT_DimensionsCheckStatistics.TooWideParcels);
	        END_IF;

	    END_REGION

	END_REGION

	REGION 11 - Button lamp

	    IF #iqUDT_EquipmentControl.Report.Stopped
	    THEN
	        #qx_ButtonLamp := FALSE;
	    END_IF;

	    IF (#iqUDT_EquipmentControl.Report.Running
	        AND NOT #iqUDT_EquipmentControl.Report.EnergySave)
	        OR (#iqUDT_EquipmentControl.Report.Dieback
	        OR #iqUDT_EquipmentControl.Report.Error)
	    THEN
	        #qx_ButtonLamp := TRUE;
	    END_IF;

	    IF #ix_ConveyorEsaveStatus
	    THEN
	        #qx_ButtonLamp := "mx_Clock_0.5Hz";
	    END_IF;

	END_REGION

	REGION 12 - Status

	    // HMI status initialization
	    #sUDT_Status.Status := 0;

	    IF #iqUDT_EquipmentControl.Report.EnergySave
	    THEN
	        #sUDT_Status.Status := "DB_HMIStatusConfiguration".EnergySave;
	    END_IF;

	    IF #iqUDT_EquipmentControl.Report.Running
	    THEN
	        #sUDT_Status.Status := "DB_HMIStatusConfiguration".Running;
	    END_IF;

	    IF #iqUDT_EquipmentControl.Report.Stopped
	    THEN
	        #sUDT_Status.Status := "DB_HMIStatusConfiguration".Stopped;
	    END_IF;

	    IF #sUDT_Status.Specific.ParcelTooHigh
	        OR #sUDT_Status.Specific.ParcelTooLong
	        OR #sUDT_Status.Specific.ParcelTooWide
	    THEN
	        #sUDT_Status.Status := "DB_HMIStatusConfiguration".DimensionError;
	    END_IF;

	    IF #iqUDT_EquipmentControl.Report.SafetyStop
	    THEN
	        #sUDT_Status.Status := "DB_HMIStatusConfiguration".SafetyStop;
	    END_IF;

	END_REGION

	REGION 13 - Update outputs

	    #qUDT_HMIStatus := #sUDT_Status;
	    #qx_Halt := #sx_Halt;
	    #qx_Lamp := #sx_Lamp;
	    #qx_WakeUp := #sx_WakeUp;
	    #qx_RunReverse := #sx_RunReverse;

	END_REGION
END_FUNCTION_BLOCK

FUNCTION_BLOCK "FB_DimensionsCheckV2"
{ S7_Optimized_Access := 'TRUE' }
VERSION : 0.1
// ATTRIBUTES
// AUTO_NUMBER = True
// BLOCK_NUMBER = 209
// END_ATTRIBUTES
   VAR_INPUT
      iUDT_DimensionsCheckConfiguration { ExternalAccessible := 'False'; ExternalVisible := 'False'; ExternalWritable := 'False'} : "UDT_DimensionsCheckConfigurationV2";   // Dimensions check configuration structure
      iUDT_DimensionsCheckCommand { ExternalAccessible := 'False'; ExternalVisible := 'False'; ExternalWritable := 'False'} : "UDT_DimensionsCheckCommandV2";   // HMI control structure
      ix_Enable { ExternalAccessible := 'False'; ExternalVisible := 'False'; ExternalWritable := 'False'} : Bool;   // TRUE -  function is active only when parcels are loaded into the system
      ix_PECBos { ExternalAccessible := 'False'; ExternalVisible := 'False'; ExternalWritable := 'False'} : Bool := TRUE;   // TRUE -  when the beginning end of section photoeye is not blocked or nothing is connected
      ix_LenghtPECLaser { ExternalAccessible := 'False'; ExternalVisible := 'False'; ExternalWritable := 'False'} : Bool;   // Length sensor - FALSE when sensor detect the parcel
      ix_MinHeightPECArray { ExternalAccessible := 'False'; ExternalVisible := 'False'; ExternalWritable := 'False'} : Bool;   // Minimum height sensor - FALSE when sensor detect the parcel
      ix_MaxHeightPEC { ExternalAccessible := 'False'; ExternalVisible := 'False'; ExternalWritable := 'False'} : Bool;   // Maximum height sensor - FALSE when sensor detect the parcel
      ii_DistanceSensor1 { ExternalAccessible := 'False'; ExternalVisible := 'False'; ExternalWritable := 'False'} : UInt;   // Distance measured by sensor between it and parcel [mm]
      ii_DistanceSensor2 { ExternalAccessible := 'False'; ExternalVisible := 'False'; ExternalWritable := 'False'} : UInt;   // Distance measured by sensor between it and parcel [mm]
      ii_Displacement { ExternalAccessible := 'False'; ExternalVisible := 'False'; ExternalWritable := 'False'} : Int;   // Conveyor displacement [cm]
      ix_Reset_Button { ExternalAccessible := 'False'; ExternalVisible := 'False'; ExternalWritable := 'False'} : Bool;   // Reset button
      ix_ReverseRunButton { ExternalAccessible := 'False'; ExternalVisible := 'False'; ExternalWritable := 'False'} : Bool;   // Reverse run button
      ix_HardwareOK { ExternalAccessible := 'False'; ExternalVisible := 'False'; ExternalWritable := 'False'} : Bool;   // TRUE when 24V on RIO with DMC signals is OK
   END_VAR

   VAR_OUTPUT
      qUDT_HMIStatus { ExternalAccessible := 'False'; ExternalVisible := 'False'; ExternalWritable := 'False'} : "UDT_DimensionsCheckStatusV2";   // Dimensions check status error structure
      qUDT_HMIData { ExternalAccessible := 'False'; ExternalVisible := 'False'; ExternalWritable := 'False'} : "UDT_DimensionsCheckHMIDataV2";   // Dimensions check HMI data structure
      qx_RequestHoldConveyor { ExternalAccessible := 'False'; ExternalVisible := 'False'; ExternalWritable := 'False'} : Bool;   // TRUE when conveyor should be stopped
      qx_RequestRunReverseConveyor { ExternalAccessible := 'False'; ExternalVisible := 'False'; ExternalWritable := 'False'} : Bool;   // TRUE when conveyor should run in reverse direction
      qx_BuzzerColumn { ExternalAccessible := 'False'; ExternalVisible := 'False'; ExternalWritable := 'False'} : Bool;   // Buzzer on column
      qx_LightColumn { ExternalAccessible := 'False'; ExternalVisible := 'False'; ExternalWritable := 'False'} : Bool;   // Light on column blue color
      qx_LightResetButton { ExternalAccessible := 'False'; ExternalVisible := 'False'; ExternalWritable := 'False'} : Bool;   // Light button blue color
   END_VAR

   VAR_IN_OUT
      iqUDT_EquipmentControl : "UDT_EquipmentControl";   // Equipment control structure
   END_VAR

   VAR
      s_HeightPEC_TimerOnOffDelay { ExternalAccessible := 'False'; ExternalVisible := 'False'; ExternalWritable := 'False'; S7_SetPoint := 'False'} : "FB_TimerOnOffDelay";   // Heigh sensor filter
      s_FB_HardwareOKSignalDelay { ExternalAccessible := 'False'; ExternalVisible := 'False'; ExternalWritable := 'False'; S7_SetPoint := 'False'} : "FB_TimerOnOffDelay";   // Hardware OK signal delay
      s_R_TRIG_ParcelTooLong {InstructionName := 'R_TRIG'; LibVersion := '1.0'; ExternalAccessible := 'False'; ExternalVisible := 'False'; ExternalWritable := 'False'; S7_SetPoint := 'False'} : R_TRIG;   // Rising edge trigger of too long parcel error
      s_R_TRIG_ParcelTooShort {InstructionName := 'R_TRIG'; LibVersion := '1.0'; ExternalAccessible := 'False'; ExternalVisible := 'False'; ExternalWritable := 'False'; S7_SetPoint := 'False'} : R_TRIG;   // Rising edge trigger of too short parcel error
      s_R_TRIG_ParcelTooHigh {InstructionName := 'R_TRIG'; LibVersion := '1.0'; ExternalAccessible := 'False'; ExternalVisible := 'False'; ExternalWritable := 'False'; S7_SetPoint := 'False'} : R_TRIG;   // Rising edge trigger of  too high parcel error
      s_R_TRIG_ParcelTooLow {InstructionName := 'R_TRIG'; LibVersion := '1.0'; ExternalAccessible := 'False'; ExternalVisible := 'False'; ExternalWritable := 'False'; S7_SetPoint := 'False'} : R_TRIG;   // Rising edge trigger of  too low parcel error
      s_R_TRIG_ParcelTooWide {InstructionName := 'R_TRIG'; LibVersion := '1.0'; ExternalAccessible := 'False'; ExternalVisible := 'False'; ExternalWritable := 'False'; S7_SetPoint := 'False'} : R_TRIG;   // Rising edge trigger of parcel too wide trigger
      s_R_TRIG_ParcelTooNarrow {InstructionName := 'R_TRIG'; LibVersion := '1.0'; ExternalAccessible := 'False'; ExternalVisible := 'False'; ExternalWritable := 'False'; S7_SetPoint := 'False'} : R_TRIG;   // Rising edge trigger of  too narrow parcel error
      s_R_TRIG_IncorrectShape {InstructionName := 'R_TRIG'; LibVersion := '1.0'; ExternalAccessible := 'False'; ExternalVisible := 'False'; ExternalWritable := 'False'; S7_SetPoint := 'False'} : R_TRIG;   // Rising edge trigger of  incorrect shape error
      s_R_TRIG_GeneralError {InstructionName := 'R_TRIG'; LibVersion := '1.0'; ExternalAccessible := 'False'; ExternalVisible := 'False'; ExternalWritable := 'False'; S7_SetPoint := 'False'} : R_TRIG;   // Rising edge trigger of general error
      s_R_TRIG_MinHeightPEC_Array {InstructionName := 'R_TRIG'; LibVersion := '1.0'; ExternalAccessible := 'False'; ExternalVisible := 'False'; ExternalWritable := 'False'; S7_SetPoint := 'False'} : R_TRIG;   // Rising edge trigger of lenght sensor
      s_R_TRIG_ResetButton {InstructionName := 'R_TRIG'; LibVersion := '1.0'; ExternalAccessible := 'False'; ExternalVisible := 'False'; ExternalWritable := 'False'; S7_SetPoint := 'False'} : R_TRIG;   // Rising edge trigger of reset button
      s_R_TRIG_ButtonOffsetDistanceSensor1 {InstructionName := 'R_TRIG'; LibVersion := '1.0'; ExternalAccessible := 'False'; ExternalVisible := 'False'; ExternalWritable := 'False'; S7_SetPoint := 'False'} : R_TRIG;   // Rising edge trigger of offset button
      s_R_TRIG_ButtonOffsetDistanceSensor2 {InstructionName := 'R_TRIG'; LibVersion := '1.0'; ExternalAccessible := 'False'; ExternalVisible := 'False'; ExternalWritable := 'False'; S7_SetPoint := 'False'} : R_TRIG;   // Rising edge trigger of offset button
      s_F_TRIG_MinHeightPEC_Array {InstructionName := 'F_TRIG'; LibVersion := '1.0'; ExternalAccessible := 'False'; ExternalVisible := 'False'; ExternalWritable := 'False'; S7_SetPoint := 'False'} : F_TRIG;   // Falling edge trigger of lenght sensor
      s_F_TRIG_WaitForAllScanData {InstructionName := 'F_TRIG'; LibVersion := '1.0'; ExternalAccessible := 'False'; ExternalVisible := 'False'; ExternalWritable := 'False'; S7_SetPoint := 'False'} : F_TRIG;   // Falling edge trigger of parcel scaned
      s_UDT_Status { ExternalAccessible := 'False'; ExternalVisible := 'False'; ExternalWritable := 'False'; S7_SetPoint := 'False'} : "UDT_DimensionsCheckStatusV2";   // Dimension check status structure
      s_UDT_DimensionsCheckStatistics { ExternalAccessible := 'False'; ExternalVisible := 'False'; ExternalWritable := 'False'; S7_SetPoint := 'False'} : "UDT_DimensionsCheckStatisticsV2";   // Dimensions check statistics
      sa_Measurement { ExternalAccessible := 'False'; ExternalVisible := 'False'; ExternalWritable := 'False'} : Array[0..200] of Struct   // Array with measurement data
         MaxHeightPEC { ExternalAccessible := 'False'; ExternalVisible := 'False'; ExternalWritable := 'False'} : Bool;
         MinHeight_Array { ExternalAccessible := 'False'; ExternalVisible := 'False'; ExternalWritable := 'False'} : Bool;
         LenghtPEC_Laser { ExternalAccessible := 'False'; ExternalVisible := 'False'; ExternalWritable := 'False'} : Bool;
         Distance_Sensor_1 { ExternalAccessible := 'False'; ExternalVisible := 'False'; ExternalWritable := 'False'} : UInt;
         Distance_Sensor_2 { ExternalAccessible := 'False'; ExternalVisible := 'False'; ExternalWritable := 'False'} : UInt;
      END_STRUCT;
      ss_Parcel { ExternalAccessible := 'False'; ExternalVisible := 'False'; ExternalWritable := 'False'} : Struct   // Structure with parcel data
         Lenght { ExternalAccessible := 'False'; ExternalVisible := 'False'; ExternalWritable := 'False'} : Int;   // Lenght [mm]
         Size { ExternalAccessible := 'False'; ExternalVisible := 'False'; ExternalWritable := 'False'} : Array[0..200] of Struct   // size arrray
            Width { ExternalAccessible := 'False'; ExternalVisible := 'False'; ExternalWritable := 'False'} : UInt;
            TooHigh { ExternalAccessible := 'False'; ExternalVisible := 'False'; ExternalWritable := 'False'} : Bool;
            TooLow { ExternalAccessible := 'False'; ExternalVisible := 'False'; ExternalWritable := 'False'} : Bool;
         END_STRUCT;
      END_STRUCT;
      ss_Positions_Distance { ExternalAccessible := 'False'; ExternalVisible := 'False'; ExternalWritable := 'False'} : Struct   // Distance is calculeted from firts sensor to the next one
         MinHeight_PEC { ExternalAccessible := 'False'; ExternalVisible := 'False'; ExternalWritable := 'False'} : Int;   // Distance between Lenght_PEC_1 and ix_MinHeightPEC [mm]
         Width_Distance_Sensor_1 { ExternalAccessible := 'False'; ExternalVisible := 'False'; ExternalWritable := 'False'} : Int;   // Distance between Lenght_PEC_1 and Width_Distance_Sensor_1 [mm]
         Width_Distance_Sensor_2 { ExternalAccessible := 'False'; ExternalVisible := 'False'; ExternalWritable := 'False'} : Int;   // Distance between Lenght_PEC_1 and Width_Distance_Sensor_2 [mm]
      END_STRUCT;
      si_CounterTooLow { ExternalAccessible := 'False'; ExternalVisible := 'False'; ExternalWritable := 'False'} : Real;   // Error detection counter - too low
      si_CounterTooHigh { ExternalAccessible := 'False'; ExternalVisible := 'False'; ExternalWritable := 'False'} : Real;   // Error detection counter - too high
      si_CounterTooWide { ExternalAccessible := 'False'; ExternalVisible := 'False'; ExternalWritable := 'False'} : Real;   // Error detection counter - too wide
      si_CounterTooNarrow { ExternalAccessible := 'False'; ExternalVisible := 'False'; ExternalWritable := 'False'} : Real;   // Error detection counter - too narrow
      si_MaxWidthParcel { ExternalAccessible := 'False'; ExternalVisible := 'False'; ExternalWritable := 'False'} : Real;   // Error detection counter - max parcel width
      sr_Tolerance { ExternalAccessible := 'False'; ExternalVisible := 'False'; ExternalWritable := 'False'} : Real;   // Tolerance used to active the error
   END_VAR
   VAR RETAIN
      si_Offset_DistanceSensor1 { ExternalAccessible := 'False'; ExternalVisible := 'False'; ExternalWritable := 'False'} : UInt;   // Distance sensor 1 offset value
      si_Offset_DistanceSensor2 { ExternalAccessible := 'False'; ExternalVisible := 'False'; ExternalWritable := 'False'} : UInt;   // Distance sensor 2 offset value
   END_VAR
   VAR
      si_ParcelLenght { ExternalAccessible := 'False'; ExternalVisible := 'False'; ExternalWritable := 'False'} : Int;   // Parcel lenght
      si_RejectDistance { ExternalAccessible := 'False'; ExternalVisible := 'False'; ExternalWritable := 'False'} : Int;   // Reject distance
      si_StatusMoveBLKVariant { ExternalAccessible := 'False'; ExternalVisible := 'False'; ExternalWritable := 'False'} : Int;   // Move BLK status
      si_DistanceToLastSensor { ExternalAccessible := 'False'; ExternalVisible := 'False'; ExternalWritable := 'False'} : Int;   // Distance to last sensor
      si_DistanceCounter { ExternalAccessible := 'False'; ExternalVisible := 'False'; ExternalWritable := 'False'} : Int;   // Distance counter used in teaching mode
      si_ParcelCounter { ExternalAccessible := 'False'; ExternalVisible := 'False'; ExternalWritable := 'False'} : Int;   // Parcel counter - count up each scaned parcel
      si_DistanceTooHighSensor { ExternalAccessible := 'False'; ExternalVisible := 'False'; ExternalWritable := 'False'} : Int;   // Distance for how long "too high sensor" is active
      si_DistanceTooLongSensor { ExternalAccessible := 'False'; ExternalVisible := 'False'; ExternalWritable := 'False'} : Int;   // Distance for how long "too long sensor" is active
      sx_ConfigurationError { ExternalAccessible := 'False'; ExternalVisible := 'False'; ExternalWritable := 'False'} : Bool;   // Configuration error
      sx_MinHeight_PEC_Filtered { ExternalAccessible := 'False'; ExternalVisible := 'False'; ExternalWritable := 'False'} : Bool;   // Filtered signal of Heigth PEC
      sx_RequestHold { ExternalAccessible := 'False'; ExternalVisible := 'False'; ExternalWritable := 'False'} : Bool;   // Static variable for hold conveyor
      sx_RequestRunReverse { ExternalAccessible := 'False'; ExternalVisible := 'False'; ExternalWritable := 'False'} : Bool;   // Run reverse request
      sx_ParcelScanning { ExternalAccessible := 'False'; ExternalVisible := 'False'; ExternalWritable := 'False'} : Bool;   // Parcel scanning in progress
      sx_ParcelScanned { ExternalAccessible := 'False'; ExternalVisible := 'False'; ExternalWritable := 'False'} : Bool;   // Parcel scanned
      sx_WaitForAllScanData { ExternalAccessible := 'False'; ExternalVisible := 'False'; ExternalWritable := 'False'} : Bool;   // Funcion is waiting for all data
      sx_NextParcelInSensorsRange { ExternalAccessible := 'False'; ExternalVisible := 'False'; ExternalWritable := 'False'} : Bool;   // Next parcel in sensors range
      sx_ParcelRejecte { ExternalAccessible := 'False'; ExternalVisible := 'False'; ExternalWritable := 'False'} : Bool;   // Parcel reject
      sx_ActiveTeachingMode { ExternalAccessible := 'False'; ExternalVisible := 'False'; ExternalWritable := 'False'} : Bool := FALSE;   // Active teaching mode
      si_RejectWindow { ExternalAccessible := 'False'; ExternalVisible := 'False'; ExternalWritable := 'False'} : Bool;   // True - when some parcel is on the sensor line
      sui_ProductWidth { ExternalAccessible := 'False'; ExternalVisible := 'False'; ExternalWritable := 'False'} : UInt;   // Product width
   END_VAR

   VAR_TEMP
      ti_LoopParcelLength : Int;   // Loop counter - Parcel length
      ti_LoopCleanArrayMeasurement : Int;   // Loop counter - Clean array measurement
      ti_LoopCleanArray : Int;   // Loop counter - Clean array
      ti_LoopErrorDetection : Int;   // Loop counter - Error detection
      ti_LoopDisplacement : Int;   // Loop counter - Displacement
      ti_ArraySize : Int;   // Array size
      ts_Position : Struct   // Sensors position
         MinHeightPEC : Int;   // PEC position
         WidthDistanceSensor1 : Int;   // Distance sensor position
         WidthDistanceSensor2 : Int;   // Distance sensor position
      END_STRUCT;
   END_VAR

   VAR CONSTANT
      ci_MeasurementArraySize : Int := 199;
   END_VAR


BEGIN
	(*
	----------------------------------------------------------------------------------------
	|                                                                                      |
	|  Copyright  2023             Fortna Europe BV                                        |
	|  All Rights Reserved         Netherlands                                             |
	|                                                                                      |
	|                                                                                      |
	----------------------------------------------------------------------------------------

	Version history:
	Date        | Version   | Author        | Remark
	----------------------------------------------------------------------------------------
	29/03/2023  | 1.0       | S. Nikodem    | First release TIA V17 | DHL Munich 2023
	15/12/2023  | 1.1       | S. Nikodem    | On site update
	04/01/2024  | 1.2       | M.Diebel      | Added "not" to "too long parcel" condition
	22/01/2024  | 1.3       | L.Klar        | New configuration error condition to avoid PLC stop
	02/02/2024  | 1.4       | R.Golonka     | Product width HMI status, HMI error status
	12/02/2024  | 1.5       | L.Klar        | Stop measuring condition changed
	12/03/2024  | 1.6       | S.Nieswiec    | Added from Munich, variable names changes according to standard

	*)

	REGION 1 - Triggers

	    // Preparating triggers for statistics.
	    #s_R_TRIG_ParcelTooLong(CLK := #s_UDT_Status.Specific.ParcelTooLongError);
	    #s_R_TRIG_ParcelTooShort(CLK := #s_UDT_Status.Specific.ParcelTooShortError);
	    #s_R_TRIG_ParcelTooHigh(CLK := #s_UDT_Status.Specific.ParcelTooHighError);
	    #s_R_TRIG_ParcelTooLow(CLK := #s_UDT_Status.Specific.ParcelTooLowError);
	    #s_R_TRIG_ParcelTooWide(CLK := #s_UDT_Status.Specific.ParcelTooWideError);
	    #s_R_TRIG_ParcelTooNarrow(CLK := #s_UDT_Status.Specific.ParcelTooNarrowError);
	    #s_R_TRIG_IncorrectShape(CLK := #s_UDT_Status.Specific.IncorrectParcelOrientationError);

	    // Sensor triggers
	    #s_R_TRIG_MinHeightPEC_Array(CLK := #sx_MinHeight_PEC_Filtered);
	    #s_F_TRIG_MinHeightPEC_Array(CLK := #sx_MinHeight_PEC_Filtered);

	    // Button trigger
	    #s_R_TRIG_ResetButton(CLK := #ix_Reset_Button);
	    #s_R_TRIG_ButtonOffsetDistanceSensor1(CLK := #iUDT_DimensionsCheckCommand.ButtonOffsetDistanceSensor1);
	    #s_R_TRIG_ButtonOffsetDistanceSensor2(CLK := #iUDT_DimensionsCheckCommand.ButtonOffsetDistanceSensor2);

	    // Parcel scaned
	    #s_F_TRIG_WaitForAllScanData(CLK := #sx_WaitForAllScanData);

	END_REGION

	REGION 2 - 24V OK signal delay

	    #s_FB_HardwareOKSignalDelay(iudi_OnDelayTime := 5000,
	                                ix_SignalToDelay := #ix_HardwareOK);

	END_REGION

	REGION 2 - Photo eye filter

	    // Minimum high check photo eye filter.
	    #s_HeightPEC_TimerOnOffDelay(iudi_OnDelayTime := #iUDT_DimensionsCheckConfiguration.PEC_Time_Delay.On_MinHeight,
	                                 iudi_OffDelayTime := #iUDT_DimensionsCheckConfiguration.PEC_Time_Delay.Off_MinHeight,
	                                 ix_SignalToDelay := NOT #ix_MinHeightPECArray,
	                                 ix_Enable := TRUE,
	                                 qx_DelayedSignal => #sx_MinHeight_PEC_Filtered);

	END_REGION

	REGION 3 - Error reset

	    // Reseting errors.
	    //
	    IF #s_R_TRIG_ResetButton.Q OR #iqUDT_EquipmentControl.Command.Reset THEN
	        #s_UDT_Status.Specific.GeneralError := False;
	    END_IF;

	    IF #s_R_TRIG_ResetButton.Q AND #si_RejectWindow
	    THEN

	        #s_UDT_Status.Specific.ParcelTooLongError := False;
	        #s_UDT_Status.Specific.ParcelTooShortError := False;
	        #s_UDT_Status.Specific.ParcelTooHighError := False;
	        #s_UDT_Status.Specific.ParcelTooLowError := False;
	        #s_UDT_Status.Specific.ParcelTooWideError := False;
	        #s_UDT_Status.Specific.ParcelTooNarrowError := False;
	        #s_UDT_Status.Specific.IncorrectParcelOrientationError := False;


	        //Check array size
	        #ti_ArraySize := "FC_GetNrOfArrayEl"(iv_Array := #sa_Measurement);

	        //Reset all data in measurement array
	        FOR #ti_LoopCleanArrayMeasurement := 0 TO (#ti_ArraySize - 1) DO

	            #sa_Measurement[#ti_LoopCleanArrayMeasurement].Distance_Sensor_1 := 0;
	            #sa_Measurement[#ti_LoopCleanArrayMeasurement].Distance_Sensor_2 := 0;
	            #sa_Measurement[#ti_LoopCleanArrayMeasurement].MaxHeightPEC := False;
	            #sa_Measurement[#ti_LoopCleanArrayMeasurement].MinHeight_Array := False;
	            #sa_Measurement[#ti_LoopCleanArrayMeasurement].LenghtPEC_Laser := False;

	        END_FOR;

	        //Check array size
	        #ti_ArraySize := "FC_GetNrOfArrayEl"(iv_Array := #ss_Parcel.Size);

	        //Reset all parcel data
	        FOR #ti_LoopCleanArray := 0 TO (#ti_ArraySize - 1) DO

	            #ss_Parcel.Size[#ti_LoopCleanArray].Width := 0;
	            #ss_Parcel.Size[#ti_LoopCleanArray].TooHigh := 0;
	            #ss_Parcel.Size[#ti_LoopCleanArray].TooLow := 0;
	            #ss_Parcel.Lenght := 0;

	        END_FOR;

	        //Reset all value after parcel reject
	        #sx_ParcelScanning := FALSE;
	        #sx_ParcelScanned := FALSE;
	        #sx_WaitForAllScanData := FALSE;
	        #sx_NextParcelInSensorsRange := FALSE;
	        #si_DistanceToLastSensor := 0;
	        #sx_RequestHold := False;
	        #sx_ParcelRejecte := False;

	    END_IF;

	END_REGION

	REGION 4 - Configuration check

	    // Save offset
	    // Offset it is a distance from sensor to side guards
	    IF #s_R_TRIG_ButtonOffsetDistanceSensor1.Q THEN
	        #si_Offset_DistanceSensor1 := #ii_DistanceSensor1;
	    END_IF;

	    IF #s_R_TRIG_ButtonOffsetDistanceSensor2.Q THEN
	        #si_Offset_DistanceSensor2 := #ii_DistanceSensor2;
	    END_IF;

	    //Copy sensors positions
	    #ts_Position.MinHeightPEC := #iUDT_DimensionsCheckConfiguration.Position.MinHeightPEC_Array / 10;
	    #ts_Position.WidthDistanceSensor1 := #iUDT_DimensionsCheckConfiguration.Position.Width_Distance_Sensor_1 / 10;
	    #ts_Position.WidthDistanceSensor2 := #iUDT_DimensionsCheckConfiguration.Position.Width_Distance_Sensor_2 / 10;

	    //Configuration check
	    #sx_ConfigurationError := #iUDT_DimensionsCheckConfiguration.Position.MinHeightPEC_Array <= 0
	    OR #iUDT_DimensionsCheckConfiguration.Position.Width_Distance_Sensor_1 <= 0
	    OR #iUDT_DimensionsCheckConfiguration.Position.Width_Distance_Sensor_2 <= 0
	    OR #iUDT_DimensionsCheckConfiguration.Position.Width_Distance_Sensor_1 >= #iUDT_DimensionsCheckConfiguration.Position.Width_Distance_Sensor_2
	    OR #si_Offset_DistanceSensor1 <= 0
	    OR #si_Offset_DistanceSensor2 <= 0;

	END_REGION

	REGION 5 - Collect data from sensors

	    IF #ix_Enable
	        AND NOT #sx_ConfigurationError
	        AND #ii_Displacement > 0
	    THEN

	        //Copy data from sensors to array
	        FOR #ti_LoopDisplacement := 1 TO #ii_Displacement DO

	            // Switch data in the array
	            #si_StatusMoveBLKVariant := MOVE_BLK_VARIANT(SRC := #sa_Measurement, COUNT := 199, SRC_INDEX := 0, DEST_INDEX := 1, DEST => #sa_Measurement);

	            //Max height PEC - Laser
	            #sa_Measurement[0].MaxHeightPEC := NOT #ix_MaxHeightPEC;

	            //Min height - RAY 26
	            #sa_Measurement[0].MinHeight_Array := NOT #ix_MinHeightPECArray;

	            //Lenght PEC - Laser
	            #sa_Measurement[0].LenghtPEC_Laser := NOT #ix_LenghtPECLaser;

	            //Distance sensor 1
	            #sa_Measurement[0].Distance_Sensor_1 := #ii_DistanceSensor1 - #si_Offset_DistanceSensor1;

	            //Distance sensor 2
	            #sa_Measurement[0].Distance_Sensor_2 := #ii_DistanceSensor2 - #si_Offset_DistanceSensor2;

	        END_FOR;

	    END_IF;

	END_REGION

	REGION 6 - Create virtual parcel

	    IF #ix_Enable
	        AND NOT #sx_ConfigurationError
	        AND NOT #sx_RequestRunReverse
	    THEN

	        //Start measuring process. Beginning of the parcel detected
	        IF
	            (#s_R_TRIG_MinHeightPEC_Array.Q OR (#sx_NextParcelInSensorsRange AND NOT #sx_ParcelScanning))
	        THEN

	            //Two parcels in the sensor range
	            #sx_NextParcelInSensorsRange := #sx_ParcelScanning;

	            //Active when parcel is detected
	            #sx_ParcelScanning := True;

	        END_IF;

	        //End of the parcel detected, wait for data from all sensors.
	        IF #s_F_TRIG_MinHeightPEC_Array.Q
	            AND #sx_ParcelScanning
	        THEN

	            #sx_ParcelScanning := False;
	            #sx_WaitForAllScanData := True;

	        END_IF;

	        //Calculate the distance to last sensor
	        IF #sx_WaitForAllScanData THEN

	            #si_DistanceToLastSensor += #ii_Displacement;

	            //Stop measuring process.
	            IF #ts_Position.WidthDistanceSensor2 <= #si_DistanceToLastSensor THEN

	                #si_DistanceToLastSensor := 0;
	                #sx_ParcelScanned := True;
	                #sx_WaitForAllScanData := False;

	                //Clean parcel data
	                FOR #ti_LoopCleanArray := 0 TO #ci_MeasurementArraySize DO

	                    #ss_Parcel.Size[#ti_LoopCleanArray].Width := 0;
	                    #ss_Parcel.Size[#ti_LoopCleanArray].TooHigh := 0;
	                    #ss_Parcel.Size[#ti_LoopCleanArray].TooLow := 0;
	                    #ss_Parcel.Lenght := 0;

	                END_FOR;

	            END_IF;

	        END_IF;

	    END_IF;

	    REGION 6.1 - Parcel calculation

	        IF #sx_ParcelScanned THEN

	            //Check array size
	            #ti_ArraySize := "FC_GetNrOfArrayEl"(iv_Array := #sa_Measurement);

	            FOR #ti_LoopParcelLength := #ts_Position.WidthDistanceSensor2 TO (#ti_ArraySize - 1) DO

	                // Length
	                IF #sa_Measurement[#ti_LoopParcelLength].MinHeight_Array THEN

	                    // Height
	                    #ss_Parcel.Size[#ss_Parcel.Lenght].TooHigh := #sa_Measurement[#ti_LoopParcelLength].MaxHeightPEC;
	                    #ss_Parcel.Size[#ss_Parcel.Lenght].TooLow := #sa_Measurement[#ti_LoopParcelLength].MinHeight_Array AND NOT #sa_Measurement[#ti_LoopParcelLength + #ts_Position.MinHeightPEC].LenghtPEC_Laser;

	                    // Width
	                    IF ((#sa_Measurement[#ti_LoopParcelLength - #ts_Position.WidthDistanceSensor1 + #ts_Position.MinHeightPEC].Distance_Sensor_1 < #iUDT_DimensionsCheckConfiguration.Position.BeltWidth)
	                        AND ((#sa_Measurement[#ti_LoopParcelLength - #ts_Position.WidthDistanceSensor2 + #ts_Position.MinHeightPEC].Distance_Sensor_2) < #iUDT_DimensionsCheckConfiguration.Position.BeltWidth))
	                    THEN
	                        #ss_Parcel.Size[#ss_Parcel.Lenght].Width :=
	                        INT_TO_UINT(#iUDT_DimensionsCheckConfiguration.Position.BeltWidth) -
	                        ((#sa_Measurement[#ti_LoopParcelLength - #ts_Position.WidthDistanceSensor1 + #ts_Position.MinHeightPEC].Distance_Sensor_1) +
	                        (#sa_Measurement[#ti_LoopParcelLength - #ts_Position.WidthDistanceSensor2 + #ts_Position.MinHeightPEC].Distance_Sensor_2));

	                        //Override overflow of UINT
	                        IF #ss_Parcel.Size[#ss_Parcel.Lenght].Width > #iUDT_DimensionsCheckConfiguration.Position.BeltWidth THEN
	                            #ss_Parcel.Size[#ss_Parcel.Lenght].Width := 0;
	                        END_IF;

	                    END_IF;

	                    #ss_Parcel.Lenght += 1;

	                END_IF;

	            END_FOR;

	            // Muliplay by 10 to have a lenght in mm
	            #ss_Parcel.Lenght *= 10;

	            //Reset data in array of measurement
	            FOR #ti_LoopCleanArrayMeasurement := #ts_Position.WidthDistanceSensor2 TO #ci_MeasurementArraySize DO

	                #sa_Measurement[#ti_LoopCleanArrayMeasurement].Distance_Sensor_1 := 0;
	                #sa_Measurement[#ti_LoopCleanArrayMeasurement].Distance_Sensor_2 := 0;
	                #sa_Measurement[#ti_LoopCleanArrayMeasurement].MaxHeightPEC := False;
	                #sa_Measurement[#ti_LoopCleanArrayMeasurement].MinHeight_Array := False;
	                #sa_Measurement[#ti_LoopCleanArrayMeasurement].LenghtPEC_Laser := False;

	            END_FOR;

	            //Only for test - Parcel counter
	            #si_ParcelCounter += 1;

	        END_IF;

	    END_REGION

	END_REGION

	REGION 7 - Error detection

	    REGION 7.1 -General Error

	        IF NOT #iUDT_DimensionsCheckCommand.DisableGeneral
	            AND #s_FB_HardwareOKSignalDelay.qx_DelayedSignal
	            AND #sx_ConfigurationError
	        THEN

	            #s_UDT_Status.Specific.GeneralError := True;

	        END_IF;

	    END_REGION

	    //Errors detection is only check when new parcel was scanned

	    //Errors counter
	    IF #sx_ParcelScanned THEN

	        //Clean counter
	        #si_CounterTooHigh := 0;
	        #si_CounterTooLow := 0;
	        #si_CounterTooWide := 0;
	        #si_CounterTooNarrow := 0;
	        #si_MaxWidthParcel := 0;

	        // Too wide parcel tolerance
	        #sr_Tolerance := INT_TO_REAL(#iUDT_DimensionsCheckConfiguration.Limit.MaxWidth) / 100 * INT_TO_REAL(#iUDT_DimensionsCheckConfiguration.Tolerance.TooWide);

	        //Value in cm
	        #si_ParcelLenght := #ss_Parcel.Lenght / 10;

	        FOR #ti_LoopErrorDetection := 1 TO #si_ParcelLenght DO

	            // Too High
	            IF #ss_Parcel.Size[#ti_LoopErrorDetection].TooHigh THEN
	                #si_CounterTooHigh += 1;
	            END_IF;
	            // Too Low
	            IF #ss_Parcel.Size[#ti_LoopErrorDetection].TooLow THEN
	                #si_CounterTooLow += 1;
	            END_IF;
	            // Too Wide
	            IF #ss_Parcel.Size[#ti_LoopErrorDetection].Width >= #iUDT_DimensionsCheckConfiguration.Limit.MaxWidth + #sr_Tolerance THEN
	                #si_CounterTooWide += 1;
	            END_IF;
	            // Too Narrow
	            IF (#ss_Parcel.Size[#ti_LoopErrorDetection].Width <= #iUDT_DimensionsCheckConfiguration.Limit.MinWidth) AND #ss_Parcel.Size[#ti_LoopErrorDetection].Width <> 0 THEN
	                #si_CounterTooNarrow += 1;
	            END_IF;
	            // Orientation detection
	            IF #si_MaxWidthParcel < #ss_Parcel.Size[#ti_LoopErrorDetection].Width THEN
	                #si_MaxWidthParcel := UINT_TO_INT(#ss_Parcel.Size[#ti_LoopErrorDetection].Width);
	            END_IF;

	        END_FOR;

	        // Tolerance
	        #si_MaxWidthParcel -= #si_MaxWidthParcel / 100.0 * INT_TO_REAL(#iUDT_DimensionsCheckConfiguration.Tolerance.Orientation);

	    END_IF;

	    REGION 7.2 - Too long parcel detection

	        //Active error when "too long" sensor is active as configured value.
	        IF NOT #ix_MinHeightPECArray
	            AND NOT #iUDT_DimensionsCheckCommand.DisableTooLongParcelError
	            AND #iUDT_DimensionsCheckConfiguration.Functionality.TooLongParcelError
	        THEN

	            #si_DistanceTooLongSensor += #ii_Displacement;

	            IF (#si_DistanceTooLongSensor * 10) > #iUDT_DimensionsCheckConfiguration.Limit.TooLongDistance THEN
	                #s_UDT_Status.Specific.ParcelTooLongError := TRUE;
	                #sx_ParcelRejecte := True;
	            END_IF;

	        ELSE
	            #si_DistanceTooLongSensor := 0;
	        END_IF;

	        IF NOT #iUDT_DimensionsCheckCommand.DisableTooLongParcelError
	            AND #sx_ParcelScanned
	            AND (#ss_Parcel.Lenght > #iUDT_DimensionsCheckConfiguration.Limit.MaxLength)
	        THEN
	            #s_UDT_Status.Specific.ParcelTooLongError := TRUE;
	            #sx_ParcelRejecte := True;
	        END_IF;

	    END_REGION

	    REGION 7.3 - Too short parcel detection

	        IF NOT #iUDT_DimensionsCheckCommand.DisableTooShortParcelError
	            AND #iUDT_DimensionsCheckConfiguration.Functionality.TooShortParcelError
	            AND #sx_ParcelScanned
	            AND (#ss_Parcel.Lenght < #iUDT_DimensionsCheckConfiguration.Limit.MinLength)
	        THEN
	            #s_UDT_Status.Specific.ParcelTooShortError := TRUE;
	            #sx_ParcelRejecte := True;
	        END_IF;

	    END_REGION

	    REGION 7.4 - Too high parcel detection

	        //Active error when "too high" sensor is active as configured value.
	        IF NOT #ix_MaxHeightPEC AND
	            NOT #iUDT_DimensionsCheckCommand.DisableTooHighParcelError
	            AND #iUDT_DimensionsCheckConfiguration.Functionality.TooHighParcelError
	        THEN

	            #si_DistanceTooHighSensor += #ii_Displacement;

	            IF (#si_DistanceTooHighSensor * 10) > #iUDT_DimensionsCheckConfiguration.Limit.TooHighDistance THEN

	                #s_UDT_Status.Specific.ParcelTooHighError := TRUE;
	                #sx_ParcelRejecte := True;

	            END_IF;

	        ELSE

	            #si_DistanceTooHighSensor := 0;

	        END_IF;

	        //Tolerance
	        #sr_Tolerance := INT_TO_REAL(#si_ParcelLenght) / 100.0 * INT_TO_REAL(#iUDT_DimensionsCheckConfiguration.Tolerance.TooHigh);

	        //Check how many times this error occurred in the array, then compare this value to tolerance.
	        //When is bigger like configured value, then set the error message.
	        IF NOT #iUDT_DimensionsCheckCommand.DisableTooHighParcelError
	            AND #sx_ParcelScanned
	            AND (#sr_Tolerance < #si_CounterTooHigh)
	        THEN
	            #s_UDT_Status.Specific.ParcelTooHighError := TRUE;
	            #sx_ParcelRejecte := True;
	        END_IF;

	    END_REGION

	    REGION 7.5 - Too low parcel detection

	        //Tolerance
	        #sr_Tolerance := INT_TO_REAL(#si_ParcelLenght) / 100.0 * INT_TO_REAL(#iUDT_DimensionsCheckConfiguration.Tolerance.TooLow);

	        //Check how many times this error occurred in the array, then compare this value to tolerance.
	        //When is bigger like configured value, then set the error message.
	        IF NOT #iUDT_DimensionsCheckCommand.DisableTooLowParcelError
	            AND #iUDT_DimensionsCheckConfiguration.Functionality.TooLowParcelError
	            AND #sx_ParcelScanned
	            AND (#sr_Tolerance < #si_CounterTooLow)
	        THEN
	            #s_UDT_Status.Specific.ParcelTooLowError := TRUE;
	            #sx_ParcelRejecte := True;
	        END_IF;

	    END_REGION

	    REGION 7.6 - Too wide parcel detection

	        //Tolerance
	        #sr_Tolerance := (INT_TO_REAL(#si_ParcelLenght) / 100.0 * INT_TO_REAL(#iUDT_DimensionsCheckConfiguration.Tolerance.TooWide));

	        //Check how many times this error occurred in the array, then compare this value to tolerance.
	        //When is bigger like configured value, then set the error message.
	        IF NOT #iUDT_DimensionsCheckCommand.DisableTooWideParcelError
	            AND #iUDT_DimensionsCheckConfiguration.Functionality.TooWideParcelError
	            AND #sx_ParcelScanned
	            AND (#sr_Tolerance < #si_CounterTooWide)
	        THEN
	            #s_UDT_Status.Specific.ParcelTooWideError := TRUE;
	            #sx_ParcelRejecte := True;
	        END_IF;

	    END_REGION

	    REGION 7.7 - Too narrow parcel detection

	        //Tolerance
	        #sr_Tolerance := INT_TO_REAL(#si_ParcelLenght) / 100.0 * INT_TO_REAL(#iUDT_DimensionsCheckConfiguration.Tolerance.TooNarrow);

	        //Check how many times this error occurred in the array, then compare this value to tolerance.
	        //When is bigger like configured value, then set the error message.
	        IF NOT #iUDT_DimensionsCheckCommand.DisableTooNarrowParcelError
	            AND #iUDT_DimensionsCheckConfiguration.Functionality.TooNarrowParcelError
	            AND #sx_ParcelScanned
	            AND (#sr_Tolerance < #si_CounterTooNarrow)
	        THEN
	            #s_UDT_Status.Specific.ParcelTooNarrowError := TRUE;
	            #sx_ParcelRejecte := True;
	        END_IF;
	    END_REGION

	    REGION 7.8 - Orientation detection

	        // Check the package position
	        IF NOT #iUDT_DimensionsCheckCommand.DisableParcelOrientationError
	            AND #iUDT_DimensionsCheckConfiguration.Functionality.ParcelOrientationError
	            AND #sx_ParcelScanned
	            AND (#ss_Parcel.Lenght < #si_MaxWidthParcel)
	        THEN
	            #s_UDT_Status.Specific.IncorrectParcelOrientationError := TRUE;
	            #sx_ParcelRejecte := True;
	        END_IF;

	    END_REGION

	    //Reset
	    #sx_ParcelScanned := false;

	END_REGION

	REGION 8 - Sequences for removing parcel

	    IF #sx_ParcelRejecte THEN

	        //To run reverse Operator must press button and BoS sensor should be free.
	        #sx_RequestRunReverse := #ix_ReverseRunButton AND #ix_PECBos;

	        #sx_RequestHold := True;
	        #si_RejectDistance -= #ii_Displacement;

	    ELSE

	        #sx_RequestRunReverse := False;
	        #si_RejectDistance := 0;

	    END_IF;

	    #si_RejectWindow := #sx_ParcelRejecte
	    AND (#si_RejectDistance > 10)
	    AND #ix_LenghtPECLaser
	    AND #ix_MinHeightPECArray
	    AND #ix_MaxHeightPEC
	    AND (#ii_DistanceSensor1 > #iUDT_DimensionsCheckConfiguration.Position.BeltWidth)
	    AND (#ii_DistanceSensor2 > #iUDT_DimensionsCheckConfiguration.Position.BeltWidth);

	END_REGION

	REGION 9 - Statistics

	    REGION 9.1 - Too long parcels statistics

	        IF #s_UDT_Status.Specific.ParcelTooLongError
	            OR #iqUDT_EquipmentControl.Command.ResetData
	        THEN
	            "FC_Statistics"(ix_Reset := #iqUDT_EquipmentControl.Command.ResetData,
	                            ix_Activate := #s_UDT_Status.Specific.ParcelTooLongError,
	                            ix_RTrigActivate := #s_R_TRIG_ParcelTooLong.Q,
	                            iqUDT_Statistics := #s_UDT_DimensionsCheckStatistics.TooLongParcels);
	        END_IF;

	    END_REGION

	    REGION 9.2 - Too short parcels statistics

	        IF #s_UDT_Status.Specific.ParcelTooShortError
	            OR #iqUDT_EquipmentControl.Command.ResetData
	        THEN
	            "FC_Statistics"(ix_Reset := #iqUDT_EquipmentControl.Command.ResetData,
	                            ix_Activate := #s_UDT_Status.Specific.ParcelTooShortError,
	                            ix_RTrigActivate := #s_R_TRIG_ParcelTooShort.Q,
	                            iqUDT_Statistics := #s_UDT_DimensionsCheckStatistics.TooShortParcels);
	        END_IF;

	    END_REGION

	    REGION 9.3 - Too high parcels statistics

	        IF #s_UDT_Status.Specific.ParcelTooHighError
	            OR #iqUDT_EquipmentControl.Command.ResetData
	        THEN
	            "FC_Statistics"(ix_Reset := #iqUDT_EquipmentControl.Command.ResetData,
	                            ix_Activate := #s_UDT_Status.Specific.ParcelTooHighError,
	                            ix_RTrigActivate := #s_R_TRIG_ParcelTooHigh.Q,
	                            iqUDT_Statistics := #s_UDT_DimensionsCheckStatistics.TooHighParcels);

	        END_IF;

	    END_REGION

	    REGION 9.4 - Too Low parcels statistics

